(* CoDeSys 2.3.9.48 project: cy-134-wg-002.pro *)
(* Libraries: Standard.lib 8.11.10 12:37:48, SYSLIBCALLBACK.LIB 8.11.10 12:37:48, Ethernet.lib 8.11.10 12:37:48, SysLibEvent.lib 8.11.10 12:37:48, SysLibFile.lib 8.11.10 12:37:48, SysLibPlcCtrl.lib 8.11.10 12:37:48, SysLibRtc.lib 8.11.10 12:37:48, SysLibSockets.lib 5.5.11 09:22:24, Util.lib 26.9.14 11:12:46, Visual.lib 8.11.10 12:37:48, WagoLibIdent.lib 25.2.13 13:49:34, WagoLibMBX_01.lib 20.3.12 16:32:38, WagoLibModbus_IP_01.lib 26.5.15 11:20:08, WagoLibStatus.lib 8.11.10 12:37:48 *)

(* PLC configuration (modules and I/O channels)
VPN_ST AT %IX0.0 [BOOLOnX_I] I 1: Digital Input
LAMP_AL AT %QX0.0 [BOOLOnX_Q] I 2: Digital Input
KEY_QE_ST AT %IX0.1 [BOOLOnX_I] I 3: Digital Input
AT %QX0.1 [BOOLOnX_Q] I 4: Digital Input
AT %IX0.2 [BOOLOnX_I] I 5: Digital Input
AT %QX0.2 [BOOLOnX_Q] I 6: Digital Input
AT %IX0.3 [BOOLOnX_I] I 7: Digital Input
AT %QX0.3 [BOOLOnX_Q] I 8: Digital Input
AT %IX0.4 [BOOLOnX_I] O 1: Digital Output
AT %QX0.4 [BOOLOnX_Q] O 2: Digital Output
AT %IX0.5 [BOOLOnX_I] O 3: Digital Output
AT %QX0.5 [BOOLOnX_Q] O 4: Digital Output
AT %IX0.6 [BOOLOnX_I] O 5: Digital Output
AT %QX0.6 [BOOLOnX_Q] O 6: Digital Output
AT %IX0.7 [BOOLOnX_I] O 7: Digital Output
AT %QX0.7 [BOOLOnX_Q] O 8: Digital Output
Fieldbus variables [FB_VARS] node 1, in %IB0 out %QB0
*)

(* Task configuration *)
TASK PLC_PRG (PRIORITY := 1); (* freewheeling *)
	PLC_PRG();
END_TASK
TASK BACnet (PRIORITY := 2, INTERVAL := T#3000ms);
	PLC_BAC();
END_TASK

(* Global variable list: Global_Constants *)
VAR_GLOBAL CONSTANT

	Plant_NAME			: STRING :='cySN:134 cyVER: Lettura sistema Desigo Ospedale Gavezzeni ';
	Plant_SN			: DWORD  :=134;	(* S/N Impianto di telecontrollo *)
	Plant_SW_VER		: WORD   :=1;		(* Versione SW installata *)


	(* Colour defines *)
	COLOR_RED			: DWORD	:= 16#2020F0;
	COLOR_YELLOW		: DWORD	:= 16#20F0F0;
	COLOR_GREEN			: DWORD	:= 16#20F020;
	COLOR_LIGHT_GREEN	: DWORD := 16#006000;

	(* Parameters *)
(*	Plant_DefaultTAmb	: INT	:=100;		(* [.1°C] Temperatura ambiente di default in caso di rottura sonda *)
	Plant_MaxRunTAmb	: INT   :=210; 		(* [.1°C] Temperatura ambiente massima funzionamento impianto *)
	Plant_AntiFreezeTAmb: INT   :=-40;		(* [.1°C] Antifreeze temperature, start circulators *)
	Plant_VRD_TAlarm	: INT   :=850; 		(* [.1°C] Temperatura di allarme VRD, blocco *)
	Plant_VRD_TMax		: INT   :=800; 		(* [.1°C] Setpoint massimo per uscita VRD *)
	Plant_VRD_TDefault	: INT	:=300;		(* [.1°C] Temperatura di default in caso di errore climatica *)
	Plant_CirOffDelay	: TIME	:=T#30m;	(* (Def.T#15m) Ritardo spegnimento pompe per ricircolo caldaia *)
	Plant_CirOnDelay	: TIME	:=T#15m;
	Plant_MaxWaterLoss	: WORD  :=2;		(* [lt/h] Massima perdita del circuito *) *)

	(* Filesystem *)
	FilesPath  			: STRING :='S:\';

	(* TCP Logger *)
	Logger_SERVER		: STRING:='';
	Logger_IP			: STRING:='10.36.201.146'; (* '192.168.100.3';*)
	Logger_PORT			: WORD  :=80;
	Logger_GETSTART		: STRING:='GET /cygmsrv/hsgm.ashx?';
	Logger_GETEND		: STRING:='$R$N$R$N';
	Logger_CHECK		: STRING:='True';
	Logger_CRLF			: STRING:='$R$N';
	Logger_DataFile		: STRING:='S:\LOG.DAT';
	Logger_DataFileOld	: STRING:='S:\LOG.BCK';
	Logger_IndexFile	: STRING:='S:\LOG.IDX';
	Logger_ConnRetries	: BYTE:=5;
	Logger_RecoverMsgs	: BYTE:=25;

	(* TCP Remote *)
	Remote_PORT			: WORD  :=10;
	Remote_WELCOME		: STRING:='Connected$R$N';
	Remote_OK			: STRING:='OK$R$N';
	Remote_ERROR		: STRING:='ERROR$R$N';

	(* TCP Sockets *)
	MAX_SEND_TCP_SERVER					 : DWORD:=30000;(*60000*)
	MAX_RECEIVE_TCP_SERVER				 : DWORD:=3000;
	MAX_RECEIVE_TCP_SERVER_SOCKET	 	 : DWORD:=1500;
	MAX_SEND_TCP_CLIENT					 : DWORD:=30000;(*15000*)
	MAX_RECEIVE_TCP_CLIENT				 : DWORD:=1500;
	MAX_RECEIVE_TCP_CLIENT_SOCKET		 : DWORD:=1500;
	MAX_RECEIVE_UDP_SERVER				 : INT  :=1472;
	MAX_RECEIVE_UDP_CLIENT				 : INT  :=1472;
	CONNECT_WATCHDOG_TIME				 : TIME :=t#10s;

END_VAR

(* Global variable list: Global_Variables *)
VAR_GLOBAL

	SYS    : typ_SYS;
	Logger : typ_Logger;


	Lamp	:	LAMP_AL_GENERALE;

	(* Analizzatori presenti  *)
	ANZ01  : obj_ANZ_Recupero_01	:= ( ID:=1 , ContabilizerMode:=0);     	(* Generale  QE1  -  Sottorete OP11 - BsB_Mulcab4_Cab4QE1 *)
	ANZ02  : obj_ANZ_Recupero_01	:= ( ID:=2 , ContabilizerMode:=0);		(* Generale  QE2 Continità - Sottorete OP11  - BsB_MulCab4_Cab4QE2C *)
	ANZ03  : obj_ANZ_Recupero_01	:= ( ID:=3 , ContabilizerMode:=0);		(* Generale  QE2  - Sottorete OP11  - BsB_MulCab4_Cab4QE2P *)
	ANZ04  : obj_ANZ_Recupero_01	:= ( ID:=4 , ContabilizerMode:=0);		(* Gruppo  Frigorifero CHW01  - Sottorete OP22  - Mult_MulC_QEGF01 *)
	ANZ05  : obj_ANZ_Recupero_01	:= ( ID:=5 , ContabilizerMode:=0);		(* Gruppo Frigorifero CHW-02 - Sottorette OP22 - Mult_MulC_QGGF02 *)
	ANZ06  : obj_ANZ_Recupero_01	:= ( ID:=6 , ContabilizerMode:=0);		(* Generale da trafo TR1 - Sottorette OP22 - Mult_QGBT02 *)
	ANZ07  : obj_ANZ_Recupero_01	:= ( ID:=7 , ContabilizerMode:=0);		(* Alimentazione Piastra 1 da QGBT - OP22 - Mult_QGBT03 *)
	ANZ08  : obj_ANZ_Recupero_01	:= ( ID:=8 , ContabilizerMode:=0);		(* Generale da trafo TR3 - OP22 - Mult_QGBT04 *)
	ANZ09  : obj_ANZ_Recupero_01	:= ( ID:=9 , ContabilizerMode:=0);		(* Gruppo frigo GF01 - OP22 - Mult_QGBT07 *)
	ANZ10  : obj_ANZ_Recupero_01	:= ( ID:=10 , ContabilizerMode:=0);	(* Riserva futuro frigorifero - OP22 - Mult_QGBT08 *)
	ANZ11  : obj_ANZ_Recupero_01	:= ( ID:=11 , ContabilizerMode:=0);	(* Riserva - OP22 - Mult_QGBT09 *)
	ANZ12  : obj_ANZ_Recupero_01	:= ( ID:=12 , ContabilizerMode:=0);	(* Riserva - OP22 - Mult_QGBT10 *)
	ANZ13  : obj_ANZ_Recupero_01	:= ( ID:=13 , ContabilizerMode:=0);	(* Impianto Water Mist - OP22 - Mult_QGBT11 *)
	ANZ14  : obj_ANZ_Recupero_01	:= ( ID:=14 , ContabilizerMode:=0);	(* QP3 Piano terzo D - OP22 - Mult_QGBT12 *)
	ANZ15  : obj_ANZ_Recupero_01	:= ( ID:=15 , ContabilizerMode:=0);	(* QP2 Piano secondo D - OP22 - Mult_QGBT13 *)
	ANZ16  : obj_ANZ_Recupero_01	:= ( ID:=16 , ContabilizerMode:=0);	(* QP1 Piano primo D - OP22 - Mult_QGBT14 *)
	ANZ17  : obj_ANZ_Recupero_01	:= ( ID:=17 , ContabilizerMode:=0);	(* QPT Piano terra D - OP22 - Mult_QGBT15 *)
	ANZ18  : obj_ANZ_Recupero_01	:= ( ID:=18 , ContabilizerMode:=0);	(* QPI Piano interrato D - OP22 - Mult_QGBT16 *)
	ANZ19  : obj_ANZ_Recupero_01	:= ( ID:=19 , ContabilizerMode:=0);	(* Alimentazione cabina ricevimento L1 - OP22 - Mult_QGBT17 *)
	ANZ20  : obj_ANZ_Recupero_01	:= ( ID:=20 , ContabilizerMode:=0);	(* Alimentazione cabina ricevimento L2 - OP22 - Mult_QGBT18 *)
	ANZ21  : obj_ANZ_Recupero_01	:= ( ID:=21 , ContabilizerMode:=0);	(*  Sezione generale da UPS1 - OP22 - Mult_QUPS01 *)
	ANZ22  : obj_ANZ_Recupero_01	:= ( ID:=22 , ContabilizerMode:=0);	(*  Sezione generale - OP22 - Mult_QUPS02 *)
	ANZ23  : obj_ANZ_Recupero_01	:= ( ID:=23 , ContabilizerMode:=0);	(*  Sezione generale da UPS2 - OP22 - Mult_QUPS03 *)
	ANZ24  : obj_ANZ_Recupero_01	:= ( ID:=24 , ContabilizerMode:=0);	(*  QP3 sezione dialisi - OP22 - Mult_QUPS04 *)
	ANZ25  : obj_ANZ_Recupero_01	:= ( ID:=25 , ContabilizerMode:=0);
	ANZ26  : obj_ANZ_Recupero_01	:= ( ID:=26 , ContabilizerMode:=0);	(* Generale Villa Elios- OP23 - Mult1'QEPC_QUPS0 *)
	ANZ27  : obj_ANZ_Recupero_01	:= ( ID:=27 , ContabilizerMode:=0);	(*Generale sez. preferenziale - OP23 - Mult1_ QGBT05*)
	ANZ28  : obj_ANZ_Recupero_01	:= ( ID:=28 , ContabilizerMode:=0);	(* generale G.E. - OP23 - Mult1'QGBT06 *)
	ANZ29  : obj_ANZ_Recupero_01	:= ( ID:=29 , ContabilizerMode:=0);	(* Gruppo frigo polivalente GP01 - OP23 - Mult1_QGBT19 *)
	ANZ30  : obj_ANZ_Recupero_01	:= ( ID:=30 , ContabilizerMode:=0);	(*QP2 quadro piano 2 - OP23 - Mul1_QGBT20*)
	ANZ31  : obj_ANZ_Recupero_01	:= ( ID:=31 , ContabilizerMode:=0);	(*QP1 quadro piano 1 - OP23 - Mult1_QGBT21*)
	ANZ32  : obj_ANZ_Recupero_01	:= ( ID:=32 , ContabilizerMode:=0);	(*QPT quadro piano terra - OP23 - Mult1_QGBT22*)
	ANZ33  : obj_ANZ_Recupero_01	:= ( ID:=33 , ContabilizerMode:=0);	(*QPI quadro piano interrato - OP23 - Mult1_QGBT23*)
	ANZ34  : obj_ANZ_Recupero_01	:= ( ID:=34 , ContabilizerMode:=0);	(*QP3 quadro piano terzo - OP23 - Mult1_QGBT24*)
	ANZ35  : obj_ANZ_Recupero_01	:= ( ID:=35 , ContabilizerMode:=0);	(*Quadro centrale UTA copertura - OP23 - Mult1_QGBT25*)
	ANZ36  : obj_ANZ_Recupero_01	:= ( ID:=36 , ContabilizerMode:=0);	(*Quadro centrale UTA esterno PT - OP23 - Mult1_QGBT26*)
	ANZ37  : obj_ANZ_Recupero_01	:= ( ID:=37 , ContabilizerMode:=0);	(*Quadro centrale idrica interrato - OP23 - Mult1_QGBT27*)
	ANZ38  : obj_ANZ_Recupero_01	:= ( ID:=38 , ContabilizerMode:=0);	(*Riserva - OP23 - Mult1_QGBT28*)
	ANZ39  : obj_ANZ_Recupero_01	:= ( ID:=39 , ContabilizerMode:=0);	(*Nuova TAC - OP23 - Mult1_QGBT29*)
	ANZ40  : obj_ANZ_Recupero_01	:= ( ID:=40 , ContabilizerMode:=0);	(*UPS1 - OP23 - Mult1_QGBT30*)
	ANZ41  : obj_ANZ_Recupero_01	:= ( ID:=41 , ContabilizerMode:=0);	(*UPS2 - OP23 - Mult1_QGBT31*)
	ANZ42  : obj_ANZ_Recupero_01	:= ( ID:=42 , ContabilizerMode:=0);	(*by-pass UPS1 - OP23 - Mult1_QGBT32*)
	ANZ43  : obj_ANZ_Recupero_01	:= ( ID:=43 , ContabilizerMode:=0);	(*by-pass UPS2 - OP23 - Mult1_QGBT33*)
	ANZ44  : obj_ANZ_Recupero_01	:= ( ID:=44 , ContabilizerMode:=0);	(*by-pass di sistema - OP23 - Mult1_QGBT34*)
	ANZ45  : obj_ANZ_Recupero_01	:= ( ID:=45 , ContabilizerMode:=0);	(*Quadro centrale termofrigorifera- OP23 - Mult1_QGBT35*)
	ANZ46  : obj_ANZ_Recupero_01	:= ( ID:=46 , ContabilizerMode:=0);			(* Gruppo Frigorifero CHW-03 - Sottorette OP22 - Mult_MulC_QGGF03 *)
	ANZ47  : obj_ANZ_Recupero_01	:= ( ID:=47 , ContabilizerMode:=0);			(* Alimentazione Piastra 1 da trafo TR1 - Sottorette OP22 - Mult_QGBT01 *)









END_VAR


VAR_GLOBAL CONSTANT


	MAX_Weekly_Schedule							: BYTE:=7;		(*Parameter for BACNET_SCHEDULE Object*)
	MAX_Exception_Schedule						: BYTE:=7;		(*Parameter for BACNET_SCHEDULE Object*)
	MAX_List_Of_Object_Property_References		: BYTE:=7;		(*Parameter for BACNET_SCHEDULE Object*)


	MAX_DateList								: BYTE:=14;	(*Parameter for BACNET_CALENDAR Object*)
	MAX_DeviceAddressBinding					: BYTE:=7;		(*Parameter for BACNET_DEVICE Object*)
	MAX_Configuration_Files						: BYTE:=4;		(*Parameter for BACNET_DEVICE Object*)
	MAX_Active_COV_Subscriptions				: BYTE:=7;		(*Parameter for BACNET_DEVICE Object*)
	MAX_List_Of_Group_Members					: BYTE:=7;		(*Parameter for BACNET_GROUP Object*)
	MAX_Accepted_Modes							: BYTE := 15;	(*Parameter for BACNET_LIFE_SAFETY_POINT / ZONE Object*)
	MAX_Life_Safety_Alarm_Values				: BYTE := 24;	(*Parameter for BACNET_LIFE_SAFETY_POINT / ZONE Object*)
	MAX_Alarm_Values							: BYTE := 24;	(*Parameter for BACNET_LIFE_SAFETY_POINT / ZONE Object*)
	MAX_Fault_Values							: BYTE := 24;	(*Parameter for BACNET_LIFE_SAFETY_POINT / ZONE Object*)
	MAX_Member_Of								: BYTE := 3;	(*Parameter for BACNET_LIFE_SAFETY_POINT / ZONE Object*)
	MAX_Zone_Members							: BYTE := 3;	(*Parameter for BACNET_LIFE_SAFETY_ ZONE Object*)
	MAX_State_Text								: BYTE:=24;	(*Parameter for BACNET_MULTISTATE_VALUE Object*)
	MAX_Alarm_Values_1							: BYTE:=24;	(*Parameter for BACNET_MULTISTATE_VALUE Object*)
	MAX_Fault_Values_1							: BYTE := 24;	(*Parameter for BACNET_MULTISTATE_VALUE Object*)
	MAX_Recipient_List							: BYTE:=8;		(*Parameter for BACNET_NOTIFICATION_CLASS Object*)
	MAX_Log_Buffer								: BYTE:=24;	(*Parameter for BACNET_TREND_LOG Object*)
	MAX_listOfPropertyReferences				: BYTE:=7;		(*Parameter for ReadAccessSpecification data type*)
END_VAR

(* Data type in Enumerationen *)
TYPE AccumulatorStatus :(
	normal_1	:=0,
	starting	:=1,
	recovered	:=2,
	abnormal	:=3,
	failed		:=4);
END_TYPE

(* Data type in Objects *)
TYPE BACNET_ACCUMULATOR :
STRUCT
	Object_Identifier			:BACnetObjectIdentifier;
	Object_Name				:STRING(48);
	Object_Type				:BACnetObjectType;
	Present_Value			:WORD;
	Description				:STRING(48);
	Device_Type				:STRING(48);
	Status_Flags				:BACnetStatusFlags;
	Event_State				:BACnetEventState;
	Reliability					:BACnetReliability;
	Out_Of_Service			:BOOL;
	Scale						:BACnetScale;
	Units						:BACnetEngineeringUnits;
	Prescale					:BACnetPrescale;
	Max_Pres_Value			:WORD;
	Value_Change_Time		:BACnetDateTime;
	Value_Before_Change	:WORD;
	Value_Set					:WORD;
	Pulse_Rate				:WORD;
	High_Limit				:WORD;
	Low_Limit					:WORD;
	Limit_Monitoring_Interval	:WORD;
	Notification_Class		:WORD;
	Time_Delay				:WORD;
	Limit_Enable				:BACnetLimitEnable;
	Event_Enable				:BACnetEventTransitionBits;
	Acked_Transitions		:BACnetEventTransitionBits;
	Notify_Type				:BACnetNotifyType;
	Event_Time_Stamps		:ARRAY [1..3] OF BACnetTimeStamp;
END_STRUCT
END_TYPE

(* Data type in Objects *)
TYPE BACNET_ANALOG_INPUT :
STRUCT
 	Object_Identifier			:BACnetObjectIdentifier;
	Object_Name				:STRING(48);
	Object_Type				:BACnetObjectType;
	Present_Value			:REAL;
	Description				:STRING(48);
	Device_Type				:STRING(48);
	Status_Flags				:BACnetStatusFlags;
	Event_State				:BACnetEventState;
	Reliability					:BACnetReliability;
	Out_of_Service			:BOOL;
	Update_Interval			:WORD;
	Units						:BACnetEngineeringUnits;
	COV_Increment			:REAL;
	Time_Delay				:WORD;
	Notification_Class		:WORD;
	High_Limit				:REAL;
	Low_Limit					:REAL;
	Deadband					:REAL;
	Limit_Enable				:BACnetLimitEnable;
	Event_Enable				:BACnetEventTransitionBits;
	Acked_Transitions		:BACnetEventTransitionBits;
	Notify_Type				:BACnetNotifyType;
	Event_Time_Stamps		:ARRAY [1..3] OF BACnetTimeStamp;
END_STRUCT
END_TYPE

(* Data type in Objects *)
TYPE BACNET_ANALOG_OUTPUT :
STRUCT
	Object_Identifier		:BACnetObjectIdentifier;
	Object_Name			:STRING(48);
	Object_Type			:BACnetObjectType;
	Present_Value		:REAL;
	Description			:STRING(48);
	Device_Type			:STRING(48);
	Status_Flags			:BACnetStatusFlags;
	Event_State			:BACnetEventState;
	Reliability				:BACnetReliability;
	Out_Of_Service		:BOOL;
	Units					:BACnetEngineeringUnits;
	Priority_Array			:BACnetPriorityArray;
	Relinquish_Default	:REAL;
	COV_Increment		:REAL;
	Time_Delay			:WORD;
	Notification_Class	:WORD;
	High_Limit			:REAL;
	Low_Limit				:REAL;
	Deadband				:REAL;
	Limit_Enable			:BACnetLimitEnable;
	Event_Enable			:BACnetEventTransitionBits;
	Acked_Transitions	:BACnetEventTransitionBits;
	Notify_Type			:BACnetNotifyType;
	Event_Time_Stamps	:ARRAY [1..3] OF BACnetTimeStamp;
END_STRUCT
END_TYPE

(* Data type in Objects *)
TYPE BACNET_ANALOG_VALUE :
STRUCT
	Object_Identifier		:BACnetObjectIdentifier;
	Object_Name			:STRING(48);
	Object_Type			:BACnetObjectType;
	Present_Value		:REAL;
	Description			:STRING(48);
	Status_Flags			:BACnetStatusFlags;
	Event_State			:BACnetEventState;
	Reliability				:BACnetReliability;
	Out_Of_Service		:BOOL;
	Units					:BACnetEngineeringUnits;
	Priority_Array			:ARRAY [1..16] OF REAL;
	Relinquish_Default	:REAL;
	COV_Increment		:REAL;
	Time_Delay			:WORD;
	Notification_Class	:WORD;
	High_Limit			:REAL;
	Low_Limit				:REAL;
	Deadband				:REAL;
	Limit_Enable			:BACnetLimitEnable;
	Event_Enable			:BACnetEventTransitionBits;
	Acked_Transitions	:BACnetEventTransitionBits;
	Notify_Type			:BACnetNotifyType;
	Event_Time_Stamps	:ARRAY [1..3] OF BACnetTimeStamp;
END_STRUCT
END_TYPE

(* Data type in Objects *)
TYPE BACNET_AVERAGING :
STRUCT
 	Object_Identifier				:BACnetObjectIdentifier;
	Object_Name					:STRING(48);
	Object_Type					:BACnetObjectType;
	Minimum_Value				:REAL;
	Minimum_Value_Timestamp:BACnetDateTime;
	Average_Value				:REAL;
	Variance_Value				:REAL;
	Maximum_Value				:REAL;
	Maximum_Value_Timestamp:BACnetDateTime;
	Description					:STRING(48);
	Attempted_Samples			:WORD;
	Valid_Samples				:WORD;
	Object_Property_Reference	:BACnetDeviceObjectPropertyReference;
	Window_Interval				:WORD;
	Window_Samples			:WORD;
END_STRUCT
END_TYPE

(* Data type in Objects *)
TYPE BACNET_BINARY_INPUT :
STRUCT
	Object_Identifier				:BACnetObjectIdentifier;
	Object_Name					:STRING(48);
	Object_Type					:BACnetObjectType;
	Present_Value				:BACnetBinaryPV;
	Description					:STRING(48);
	Device_Type					:STRING(48);
	Status_Flags					:BACnetStatusFlags;
	Event_State					:BACnetEventState;
	Reliability						:BACnetReliability;
	Out_Of_Service				:BOOL;
	Polarity						:BACnetPolarity;
	Inactive_Text					:STRING(48);
	Active_Text					:STRING(48);
	Change_Of_State_Time		:BACnetDateTime;
	Change_Of_State_Count		:WORD;
	Time_Of_State_Count_Reset:BACnetDateTime;
	Elapsed_Active_Time			:DWORD;
	Time_Of_Active_Time_Reset:BACnetDateTime;
	Time_Delay					:WORD;
	Notification_Class			:WORD;
	Alarm_Value					:BACnetBinaryPV;
	Event_Enable					:BACnetEventTransitionBits;
	Acked_Transitions			:BACnetEventTransitionBits;
	Notify_Type					:BACnetNotifyType;
	Event_Time_Stamps			:ARRAY [1..3] OF BACnetTimeStamp;
END_STRUCT
END_TYPE

(* Data type in Objects *)
TYPE BACNET_BINARY_OUTPUT :
STRUCT
 Object_Identifier					:BACnetObjectIdentifier;
 Object_Name						:STRING(48);
 Object_Type						:BACnetObjectType;
 Present_Value					:BACnetBinaryPV;
 Description						:STRING(48);
 Device_Type						:STRING(48);
 Status_Flags						:BACnetStatusFlags;
 Event_State						:BACnetEventState;
 Reliability							:BACnetReliability;
 Out_Of_Service					:BOOL;
 Polarity							:BACnetPolarity;
 Inactive_Text						:STRING(48);
 Active_Text						:STRING(48);
 Change_Of_State_Time			:BACnetDateTime;
 Change_Of_State_Count		:WORD;
 Time_Of_State_Count_Reset	:BACnetDateTime;
 Elapsed_Active_Time			:DWORD;
 Time_Of_Active_Time_Reset	:BACnetDateTime;
 Minimum_Off_Time				:DWORD;
 Minimum_On_Time				:DWORD;
 Priority_Array						:BACnetPriorityArray;
 Relinquish_Default				:BACnetBinaryPV;
 Time_Delay						:WORD;
 Notification_Class				:WORD;
 Feedback_Value					:BACnetBinaryPV;
 Event_Enable						:BACnetEventTransitionBits;
 Acked_Transitions				:BACnetEventTransitionBits;
 Notify_Type						:BACnetNotifyType;
 Event_Time_Stamps				:ARRAY [1..3] OF BACnetTimeStamp;
END_STRUCT
END_TYPE

(* Data type in Objects *)
TYPE BACNET_BINARY_VALUE :
STRUCT
	Object_Identifier					:BACnetObjectIdentifier;
	Object_Name						:STRING(48);
	Object_Type						:BACnetObjectType;
	Present_Value					:BACnetBinaryPV;
	Description						:STRING(48);
	Status_Flags						:BACnetStatusFlags;
	Event_State						:BACnetEventState;
	Reliability							:BACnetReliability;
	Out_Of_Service					:BOOL;
	Inactive_Text						:STRING(48);
	Active_Text						:STRING(48);
	Change_Of_State_Time			:BACnetDateTime;
	Change_Of_State_Count			:DWORD;
	Time_Of_State_Count_Reset	:BACnetDateTime;
	Elapsed_Active_Time				:DWORD;
	Time_Of_Active_Time_Reset	:BACnetDateTime;
	Minimum_Off_Time				:DWORD;
	Minimum_On_Time				:DWORD;
	Priority_Array						:ARRAY [1..16] OF BACnetBinaryPV;
	Relinquish_Default				:BACnetBinaryPV;
	Time_Delay						:WORD;
	Notification_Class				:WORD;
	Alarm_Value						:BACnetBinaryPV;
	Event_Enable						:BACnetEventTransitionBits;
	Acked_Transitions				:BACnetEventTransitionBits;
	Notify_Type						:BACnetNotifyType;
	Event_Time_Stamps				:ARRAY [1..3] OF BACnetTimeStamp;
END_STRUCT
END_TYPE

(* Data type in Objects *)
TYPE BACNET_CALENDAR :
STRUCT
	Object_Identifier		:BACnetObjectIdentifier;
	Object_Name			:STRING(48);
	Object_Type			:BACnetObjectType;
	Description			:STRING(48);
	Present_Value		:BOOL;
	Date_List				:ARRAY[0..MAX_DateList] OF BACnetCalendarEntry;
END_STRUCT
END_TYPE

(* Data type in Objects *)
TYPE BACNET_COMMAND :
STRUCT
	Object_Identifier			:BACnetObjectIdentifier;
	Object_Name				:STRING(48);
	Object_Type				:BACnetObjectType;
	Description				:STRING(48);
	Present_Value			:WORD;
	In_Process				:BOOL;
	All_Writes_Successful	:BOOL;
	Action_					:ARRAY [1..3] OF BACnetActionList;
	Action_Text				:ARRAY [1..3] OF STRING(48);
END_STRUCT
END_TYPE

(* Data type in Objects *)
TYPE BACNET_DEVICE :
STRUCT
	Object_Identifier						:BACnetObjectIdentifier;
	Object_Name							:STRING(48);
	Object_Type							:BACnetObjectType;
	System_Status						:BACnetDeviceStatus;
	Vendor_Name						:STRING(48);
	Vendor_Identifier						:WORD;
	Model_Name							:STRING(48);
	Firmware_Revision					:STRING(48);
	Application_Software_Version		:STRING(48);
	Location								:STRING(48);
	Description							:STRING(48);
	Protocol_Version						:WORD;
	Protocol_Revision					:WORD;
	Protocol_Services_Supported		:BACnetServicesSupported;
	Protocol_Object_Types_Supported	:BACnetObjectTypesSupported;
	Object_List							:ARRAY [1..3] OF BACnetObjectIdentifier;
	Max_APDU_Length_Accepted		:WORD;
	Segmentation_Supported			:BACnetSegmentation;
	Max_Segments_Accepted			:WORD;
	Local_Time							:TIME;
	Local_Date							:DATE;
	UTC_Offset							:INT;
	Daylight_Savings_Status				:BOOL;
	APDU_Segment_Timeout			:WORD;
	APDU_Timeout						:WORD;
	Number_Of_APDU_Retries			:WORD;
	Device_Address_Binding				:ARRAY [0..MAX_DeviceAddressBinding] OF BACnetAddressBinding;
	Database_Revision					:WORD;
	Configuration_Files					:ARRAY [1..MAX_Configuration_Files] OF BACnetObjectIdentifier;
	Last_Restore_Time					:BACnetTimeStamp;
	Backup_Failure_Timeout				:WORD;
	Active_COV_Subscriptions			:ARRAY [0..MAX_Active_COV_Subscriptions] OF BACnetCOVSubscription;
END_STRUCT
END_TYPE

(* Data type in Objects *)
TYPE BACNET_EVENT_ENROLLMENT :
STRUCT
	Object_Identifier				:BACnetObjectIdentifier;
	Object_Name					:STRING(48);
	Object_Type					:BACnetObjectType;
	Description					:STRING(48);
	Event_Type					:BACnetEventType;
	Notify_Type					:BACnetNotifyType;
	Event_Parameters			:BACnetEventParameter;
	Object_Property_Reference	:BACnetDeviceObjectPropertyReference;
	Event_State					:BACnetEventState;
	Event_Enable					:BACnetEventTransitionBits;
	Acked_Transitions			:BACnetEventTransitionBits;
	Notification_Class			:WORD;
	Event_Time_Stamps			:ARRAY [1..3] OF BACnetTimeStamp;
END_STRUCT
END_TYPE

(* Data type in Objects *)
TYPE BACNET_FILE :
STRUCT
	Object_Identifier		:BACnetObjectIdentifier;
	Object_Name			:STRING(48);
	Object_Type			:BACnetObjectType;
	Description			:STRING(48);
	File_Type				:STRING(48);
	File_Size				:WORD;
	Modification_Date		:BACnetDateTime;
	Archive					:BOOL;
	Read_Only_			:BOOL;
	File_Access_Method	:BACnetFileAccessMethod;
END_STRUCT
END_TYPE

(* Data type in Objects *)
TYPE BACNET_GROUP :
STRUCT
	Object_Identifier			:BACnetObjectIdentifier;
	Object_Name				:STRING(48);
	Object_Type				:BACnetObjectType;
	Description				:STRING(48);
	List_Of_Group_Members	:ARRAY [0..MAX_List_Of_Group_Members] OF ReadAccessSpecification;
	Present_Value			:ARRAY [0..MAX_List_Of_Group_Members] OF ReadAccessResult;
END_STRUCT
END_TYPE

(* Data type in Objects *)
TYPE BACNET_LIFE_SAFETY_POINT :
STRUCT
	Object_Identifier				:BACnetObjectIdentifier;
	Object_Name					:STRING(48);
	Object_Type					:BACnetObjectType;
	Present_Value				:BACnetLifeSafetyState;
	Tracking_Value				:BACnetLifeSafetyState;
	Description					:STRING(48);
	Device_Type					:STRING(48);
	Status_Flags					:BACnetStatusFlags;
	Event_State					:BACnetEventState;
	Reliability						:BACnetReliability;
	Out_Of_Service				:BOOL;
	Mode							:BACnetLifeSafetyMode;
	Accepted_Modes				:ARRAY [0..MAX_Accepted_Modes] OF BACnetLifeSafetyMode;
	Time_Delay					:WORD;
	Notification_Class			:WORD;
	Life_Safety_Alarm_Values	:ARRAY  [0..MAX_Life_Safety_Alarm_Values]  OF BACnetLifeSafetyState;
	Alarm_Values					:ARRAY  [0..MAX_Alarm_Values]  OF BACnetLifeSafetyState;
	Fault_Values					:ARRAY  [0..MAX_Fault_Values]  OF BACnetLifeSafetyState;
	Event_Enable					:BACnetEventTransitionBits;
	Acked_Transitions			:BACnetEventTransitionBits;
	Notify_Type					:BACnetNotifyType;
	Event_Time_Stamps			:ARRAY [1..3] OF BACnetTimeStamp;
	Silenced						:BACnetSilencedState;
	Operation_Expected			:BACnetLifeSafetyOperation;
	Maintenance_Required		:BACnetMaintenance;
	Setting							:BYTE;
	Direct_Reading				:REAL;
	Units							:BACnetEngineeringUnits;
	Member_Of					:ARRAY [1..MAX_Member_Of]  OF BACnetDeviceObjectReference;
END_STRUCT
END_TYPE

(* Data type in Objects *)
TYPE BACNET_LIFE_SAFETY_ZONE :
STRUCT
	Object_Identifier				:BACnetObjectIdentifier;
	Object_Name					:STRING(48);
	Object_Type					:BACnetObjectType;
	Present_Value				:BACnetLifeSafetyState;
	Tracking_Value				:BACnetLifeSafetyState;
	Description					:STRING(48);
	Device_Type					:STRING(48);
	Status_Flags					:BACnetStatusFlags;
	Event_State					:BACnetEventState;
	Reliability						:BACnetReliability;
	Out_Of_Service				:BOOL;
	Mode							:BACnetLifeSafetyMode;
	Accepted_Modes				:ARRAY  [0..MAX_Accepted_Modes] OF BACnetLifeSafetyMode;
	Time_Delay					:WORD;
	Notification_Class			:WORD;
	Life_Safety_Alarm_Values	:ARRAY [0..MAX_Life_Safety_Alarm_Values] OF BACnetLifeSafetyState;
	Alarm_Values					:ARRAY [0..MAX_Alarm_Values] OF BACnetLifeSafetyState;
	Fault_Values					:ARRAY [0..MAX_Fault_Values] OF BACnetLifeSafetyState;
	Event_Enable					:BACnetEventTransitionBits;
	Acked_Transitions			:BACnetEventTransitionBits;
	Notify_Type					:BACnetNotifyType;
	Event_Time_Stamps			:ARRAY [1..3] OF BACnetTimeStamp;
	Silenced						:BACnetSilencedState;
	Operation_Expected			:BACnetLifeSafetyOperation;
	Maintenance_Required		:BOOL;
	Zone_Members				:ARRAY [1..MAX_Zone_Members] OF BACnetDeviceObjectReference;
	Member_Of					:ARRAY [1..MAX_Member_Of] OF BACnetDeviceObjectReference;
END_STRUCT
END_TYPE

(* Data type in Objects *)
TYPE BACNET_LOOP :
STRUCT
	Object_Identifier						:BACnetObjectIdentifier;
	Object_Name							:STRING(48);
	Object_Type							:BACnetObjectType;
	Present_Value						:REAL;
	Description							:STRING(48);
	Status_Flags							:BACnetStatusFlags;
	Event_State							:BACnetEventState;
	Reliability								:BACnetReliability;
	Out_Of_Service						:BOOL;
	Update_Interval						:WORD;
	Output_Units							:BACnetEngineeringUnits;
	Manipulated_Variable_Reference	:BACnetObjectPropertyReference;
	Controlled_Variable_Reference		:BACnetObjectPropertyReference;
	Controlled_Variable_Value			:REAL;
	Controlled_Variable_Units			:BACnetEngineeringUnits;
	Setpoint_Reference					:BACnetSetpointReference;
	Setpoint								:REAL;
	ACTION_								:BACnetAction;
	Proportional_Constant				:REAL;
	Proportional_Constant_Units		:BACnetEngineeringUnits;
	Integral_Constant						:REAL;
	Integral_Constant_Units				:BACnetEngineeringUnits;
	Derivative_Constant					:REAL;
	Derivative_Constant_Units			:BACnetEngineeringUnits;
	Bias									:REAL;
	Maximum_Output						:REAL;
	Minimum_Output						:REAL;
	Priority_For_Writing					:WORD;
	COV_Increment						:REAL;
	Time_Delay							:WORD;
	Notification_Class					:WORD;
	Error_Limit							:REAL;
	Event_Enable							:BACnetEventTransitionBits;
	Acked_Transitions					:BACnetEventTransitionBits;
	Notify_Type							:BACnetNotifyType;
	Event_Time_Stamps					:ARRAY [1..3] OF BACnetTimeStamp;
END_STRUCT
END_TYPE

(* Data type in Objects *)
TYPE BACNET_MULTISTATE_VALUE :
STRUCT
	Object_Identifier		:BACnetObjectIdentifier;
	Object_Name			:STRING(48);
	Object_Type			:BACnetObjectType;
	Present_Value		:WORD;
	Description			:STRING(48);
	Status_Flags			:BACnetStatusFlags;
	Event_State			:BACnetEventState;
	Reliability				:BACnetReliability;
	Out_Of_Service		:BOOL;
	Number_Of_States	:WORD;
	State_Text				:ARRAY [1..MAX_State_Text] OF STRING(48);
	Priority_Array			:BACnetPriorityArray;
	Relinquish_Default	:WORD;
	Time_Delay			:WORD;
	Notification_Class	:WORD;
	Alarm_Values			:ARRAY [1..MAX_Alarm_Values_1] OF WORD;
	Fault_Values			:ARRAY [1..MAX_Fault_Values_1] OF WORD;
	Event_Enable			:BACnetEventTransitionBits;
	Acked_Transitions	:BACnetEventTransitionBits;
	Notify_Type			:BACnetNotifyType;
	Event_Time_Stamps	:ARRAY [1..3] OF BACnetTimeStamp;
END_STRUCT
END_TYPE

(* Data type in Objects *)
TYPE BACNET_NOTIFICATION_CLASS :
STRUCT
	Object_Identifier		:BACnetObjectIdentifier;
	Object_Name			:STRING(48);
	Object_Type			:BACnetObjectType;
	Description			:STRING(48);
	Notification_Class	:WORD;
	Priority					:ARRAY [1..3] OF WORD;
	Ack_Required			:BACnetEventTransitionBits;
	Recipient_List			:ARRAY [0..MAX_Recipient_List] OF BACnetDestination;
END_STRUCT
END_TYPE

(* Data type in Objects *)
TYPE BACNET_PROGRAM :
STRUCT
	Object_Identifier			:BACnetObjectIdentifier;
	Object_Name				:STRING(48);
	Object_Type				:BACnetObjectType;
	Program_State			:BACnetProgramState;
	Program_Change			:BACnetProgramRequest;
	Reason_For_Halt			:BACnetProgramError;
	Description_Of_Halt		:STRING(48);
 	Program_Location		:STRING(48);
	Description				:STRING(48);
	Status_Flags				:BACnetStatusFlags;
	Reliability					:BACnetReliability;
	Out_Of_Service			:BOOL;
END_STRUCT
END_TYPE

(* Data type in Objects *)
TYPE BACNET_PULSE_CONVERTER :
STRUCT
	Object_Identifier			:BACnetObjectIdentifier;
	Object_Name				:STRING(48);
	Object_Type				:BACnetObjectType;
	Description				:STRING(48);
	Present_Value			:REAL;
	Input_Reference			:BACnetObjectPropertyReference;
	Status_Flags				:BACnetStatusFlags;
	Event_State				:BACnetEventState;
	Reliability					:BACnetReliability;
	Out_Of_Service			:BOOL;
	Units						:BACnetEngineeringUnits;
	Scale_Factor				:REAL;
	Adjust_Value				:REAL;
	Count						:WORD;
	Update_Time				:BACnetDateTime;
	Count_Change_Time		:BACnetDateTime;
	Count_Before_Change	:WORD;
	COV_Increment			:REAL;
	COV_Period				:WORD;
	Notification_Class		:WORD;
	Time_Delay				:WORD;
	High_Limit				:REAL;
	Low_Limit					:REAL;
	Deadband					:REAL;
	Limit_Enable				:BACnetLimitEnable;
	Event_Enable				:BACnetEventTransitionBits;
	Acked_Transitions		:BACnetEventTransitionBits;
	Notify_Type				:BACnetNotifyType;
	Event_Time_Stamps		:ARRAY [1..3] OF BACnetTimeStamp;
END_STRUCT
END_TYPE

(* Data type in Objects *)
TYPE BACNET_SCHEDULE :
STRUCT
	Object_Identifier							:BACnetObjectIdentifier;
	Object_Name								:STRING(48);
	Object_Type								:BACnetObjectType;
	Present_Value							:BACnetAny;
	Description								:STRING(48);
	Effective_Period							:BACnetDateRange;
	Weekly_Schedule							:ARRAY [0..MAX_Weekly_Schedule] OF BACnetDailySchedule;
	Exception_Schedule						:ARRAY [0..MAX_Exception_Schedule] OF BACnetSpecialEvent;
	Schedule_Default							:BACnetAny;
	List_Of_Object_Property_References	:ARRAY [0..MAX_List_Of_Object_Property_References] OF BACnetDeviceObjectPropertyReference;
	Priority_For_Writing						:BYTE;
	Status_Flags								:BACnetStatusFlags;
	Reliability									:BACnetReliability;
	Out_Of_Service							:BOOL;
END_STRUCT
END_TYPE

(* Data type in Objects *)
TYPE BACNET_TREND_LOG :
STRUCT
	Object_Identifier				:BACnetObjectIdentifier;
	Object_Name					:STRING(48);
	Object_Type					:BACnetObjectType;
	Description					:STRING(48);
	Log_Enable					:BOOL;
	Start_Time					:BACnetDateTime;
	Stop_Time					:BACnetDateTime;
	Log_DeviceObjectProperty	:BACnetDeviceObjectPropertyReference;
	Log_Interval					:WORD;
	COV_Resubscription_Interval:WORD;
	Client_COV_Increment		:BACnetClientCOV;
	Stop_When_Full				:BOOL;
	Buffer_Size					:DWORD;
	Log_Buffer					:ARRAY [0..MAX_Log_Buffer] OF BACnetLogRecord;
	Record_Count				:DWORD;
	Total_Record_Count			:DWORD;
	Notification_Threshold		:DWORD;
	Records_Since_Notification	:DWORD;
	Last_Notify_Record			:DWORD;
	Event_State					:BACnetEventState;
	Notification_Class			:WORD;
	Event_Enable					:BACnetEventTransitionBits;
	Acked_Transitions			:BACnetEventTransitionBits;
	Notify_Type					:BACnetNotifyType;
	Event_Time_Stamps			:ARRAY [1..3] OF BACnetTimeStamp;
END_STRUCT
END_TYPE

(* Data type in Datatypes *)
TYPE BACnetAccumulatorRecord :
STRUCT
	timestamp 			:BACnetDateTime;
	presentValue 			:WORD;
	accumulatedValue 	:WORD;
	accumulatorStatus	:AccumulatorStatus;
END_STRUCT
END_TYPE

(* Data type in Enumerationen *)
TYPE BACnetAction :(
	direct		:=0,
	reverse	:=1);
END_TYPE

(* Data type in Datatypes *)
TYPE BACnetActionCommand :
STRUCT
	deviceIdentifier		:BACnetObjectIdentifier;
	objectIdentifier		:BACnetObjectIdentifier;
	propertyIdentifier		:BACnetPropertyIdentifier;
	propertyArrayIndex	:WORD;
	priority					:WORD;
	postDelay				:WORD;
	quitOnFailure			:BOOL;
	writeSuccessful		:BOOL;
END_STRUCT
END_TYPE

(* Data type in Datatypes *)
TYPE BACnetActionList :
STRUCT
	BACnetAction : BACnetActionCommand;
END_STRUCT
END_TYPE

(* Data type in Datatypes *)
TYPE BACnetAddress :
STRUCT
	network_number	:WORD;
	mac_address		:BYTE;
END_STRUCT
END_TYPE

(* Data type in Datatypes *)
TYPE BACnetAddressBinding :
STRUCT
	deviceObjectIdentifier		:BACnetObjectIdentifier;
	deviceAddress			:BACnetAddress;
END_STRUCT
END_TYPE

(* Data type in Datatypes/internal *)
TYPE BACnetAny :
STRUCT
	CHOICE	:WORD;
	SIZE		:BYTE;
	VALUE		:ARRAY [0..254] OF BYTE;
END_STRUCT
END_TYPE

(* Data type in Enumerationen *)
TYPE BACnetBinaryPV :(
	inactive	:=0,
	active		:=1);
END_TYPE

(* Data type in Datatypes *)
TYPE BACnetCalendarEntry :
STRUCT
	CHOICE	:BYTE;
	VALUE		:ARRAY [0..21] OF BYTE;
END_STRUCT
END_TYPE

(* Data type in Datatypes *)
TYPE BACnetClientCOV :
STRUCT
	CHOICE	:BYTE;
	VALUE		:REAL;
END_STRUCT
END_TYPE

(* Data type in Datatypes *)
TYPE BACnetCOVSubscription :
STRUCT
	Recipient						:BACnetRecipientProcess;
	MonitoredPropertyReference	:BACnetObjectPropertyReference;
	IssueConfirmedNotifications	:BOOL;
	TimeRemaining				:WORD;
	COVIncrement				:REAL;
END_STRUCT
END_TYPE

(* Data type in Datatypes *)
TYPE BACnetDailySchedule :
STRUCT
	count			:WORD;
	day_schedule	:BACnetTimeValue;
END_STRUCT
END_TYPE

(* Data type in Datatypes *)
TYPE BACnetDateRange :
STRUCT
	StartDate		:DATE;
	endDate		:DATE;
END_STRUCT
END_TYPE

(* Data type in Datatypes *)
TYPE BACnetDateTime :
STRUCT
	BACnetDate	:DATE;
	BACnetTime	:TOD;
END_STRUCT
END_TYPE

(* Data type in Datatypes *)
TYPE BACnetDaysOfWeek :
STRUCT
	monday		:BOOL;
	tuesday		:BOOL;
	wednesday	:BOOL;
	thursday		:BOOL;
	friday			:BOOL;
	saturday		:BOOL;
	sunday		:BOOL;
END_STRUCT
END_TYPE

(* Data type in Datatypes *)
TYPE BACnetDestination :
STRUCT
	validDays						:BACnetDaysOfWeek;
	fromTime						:TIME;
	toTime							:TIME;
	recipient						:BACnetRecipient;
	processIdentifier				:DWORD;
	issueConfirmedNotifications	:BOOL;
	transitions						:BACnetEventTransitionBits;
END_STRUCT
END_TYPE

(* Data type in Datatypes *)
TYPE BACnetDeviceObjectPropertyReference :
STRUCT
	objectIdentifier		:BACnetObjectIdentifier;
	propertyIdentifier		:BACnetPropertyIdentifier;
	propertyArrayIndex	:WORD;
	deviceIdentifier		:BACnetObjectIdentifier;
	devicePresent			:BOOL;
END_STRUCT
END_TYPE

(* Data type in Datatypes *)
TYPE BACnetDeviceObjectPropertyValue :
STRUCT
	deviceIdentifier	: BACnetObjectIdentifier;
	objectIdentifier	: BACnetObjectIdentifier;
	propertyIdentifier 	: BACnetPropertyIdentifier;
	arrayIndex 			:WORD;
END_STRUCT
END_TYPE

(* Data type in Datatypes *)
TYPE BACnetDeviceObjectReference :
STRUCT
	deviceIdentifier	:BACnetObjectIdentifier;
	objectIdentifier	:BACnetObjectIdentifier;
	devicePresent		:BOOL;
END_STRUCT
END_TYPE

(* Data type in Enumerationen *)
TYPE BACnetDeviceStatus :(
	operational				:=0,
	operational_read_only	:=1,
	download_required		:=2,
	download_in_progress	:=3,
	non_operational			:=4,
	backup_in_progress		:=5);
END_TYPE

(* Data type in Enumerationen *)
TYPE BACnetEngineeringUnits :(
	square_meters	:=	0	,
	square_feet		:=	1	,
	milliamperes		:=	2	,
	amperes			:=	3	,
	ohms				:=	4	,
	volts				:=	5	,
	kilovolts			:=	6	,
	megavolts			:=	7	,
	volt_amperes		:=	8	,
	kilovolt_amperes	:=	9	,
	megavolt_amperes			:=	10	,
	volt_amperes_reactive		:=	11	,
	kilovolt_amperes_reactive	:=	12	,
	megavolt_amperes_reactive	:=	13	,
	degrees_phase				:=	14	,
	power_factor					:=	15	,
	joules							:=	16	,
	kilojoules					:=	17	,
	watt_hours				:=	18	,
	kilowatt_hours			:=	19	,
	btus						:=	20	,
	therms						:=	21	,
	ton_hours					:=	22	,
	joules_per_kilogram_dry_air		:=	23	,
	btus_per_pound_dry_air			:=	24	,
	cycles_per_hour					:=	25	,
	cycles_per_minute				:=	26	,
	hertz								:=	27	,
	grams_of_water_per_kilogram_dry_air	:=	28	,
	percent_relative_humidity				:=	29	,
	millimeters								:=	30	,
	meters			:=	31	,
	inches			:=	32	,
	feet			:=	33	,
	watts_per_square_foot		:=	34	,
	watts_per_square_meter		:=	35	,
	lumens						:=	36	,
	luxes							:=	37	,
	foot_candles				:=	38	,
	kilograms					:=	39	,
	pounds_mass			:=	40	,
	tons						:=	41	,
	kilograms_per_second	:=	42	,
	kilograms_per_minute	:=	43	,
	kilograms_per_hour		:=	44	,
	pounds_mass_per_minute	:=	45	,
	pounds_mass_per_hour	:=	46	,
	watts			:=	47	,
	kilowatts		:=	48	,
	megawatts	:=	49	,
	btus_per_hour	:=	50	,
	horsepower		:=	51	,
	tons_refrigeration	:=	52	,
	pascals			:=	53	,
	kilopascals		:=	54	,
	bars				:=	55	,
	pounds_force_per_square_inch	:=	56	,
	centimeters_of_water		:=	57	,
	inches_of_water			:=	58	,
	millimeters_of_mercury	:=	59	,
	centimeters_of_mercury	:=	60	,
	inches_of_mercury		:=	61	,
	degrees_Celsius			:=	62	,
	degrees_Kelvin			:=	63	,
	degrees_Fahrenheit		:=	64	,
	degree_days_Celsius	:=	65	,
	degree_days_Fahrenheit	:=	66	,
	years		:=	67	,
	months	:=	68	,
	weeks		:=	69	,
	days		:=	70	,
	hours		:=	71	,
	minutes	:=	72	,
	seconds	:=	73	,
	meters_per_second	:=	74	,
	kilometers_per_hour	:=	75	,
	feet_per_second		:=	76	,
	feet_per_minute		:=	77	,
	miles_per_hour		:=	78	,
	cubic_feet				:=	79	,
	cubic_meters			:=	80	,
	imperial_gallons		:=	81	,
	liters					:=	82	,
	us_gallons			:=	83	,
	cubic_feet_per_minute		:=	84	,
	cubic_meters_per_second	:=	85	,
	imperial_gallons_per_minute	:=	86	,
	liters_per_second				:=	87	,
	liters_per_minute					:=	88	,
	us_gallons_per_minute			:=	89	,
	degrees_angular					:=	90	,
	degrees_Celsius_per_hour		:=	91	,
	degrees_Celsius_per_minute	:=	92	,
	degrees_Fahrenheit_per_hour	:=	93	,
	degrees_Fahrenheit_per_minute	:=	94	,
	no_units				:=	95	,
	parts_per_million		:=	96	,
	parts_per_billion		:=	97	,
	percent				:=	98	,
	percent_per_second	:=	99	,
	per_minute			:=	100	,
	per_second			:=	101	,
	psi_per_degree_Fahrenheit	:=	102	,
	radians					:=	103	,
	revolutions_per_minute	:=	104	,
	currency1					:=	105	,
	currency2					:=	106	,
	currency3					:=	107	,
	currency4					:=	108	,
	currency5					:=	109	,
	currency6					:=	110	,
	currency7					:=	111	,
	currency8					:=	112	,
	currency9					:=	113	,
	currency10				:=	114	,
	square_inches			:=	115	,
	square_centimeters		:=	116	,
	btus_per_pound			:=	117	,
	centimeters				:=	118	,
	pounds_mass_per_second	:=	119	,
	delta_degrees_Fahrenheit	:=	120	,
	delta_degrees_Kelvin		:=	121	,
	kilohms					:=	122	,
	megohms					:=	123	,
	millivolts					:=	124	,
	kilojoules_per_kilogram	:=	125	,
	megajoules				:=	126	,
	joules_per_degree_Kelvin				:=	127	,
	joules_per_kilogram_degree_Kelvin	:=	128	,
	kilohertz			:=	129	,
	megahertz			:=	130	,
	per_hour			:=	131	,
	milliwatts			:=	132	,
	hectopascals		:=	133	,
	millibars			:=	134	,
	cubic_meters_per_hour	:=	135	,
	liters_per_hour			:=	136	,
	kilowatt_hours_per_square_meter	:=	137	,
	kilowatt_hours_per_square_foot		:=	138	,
	megajoules_per_square_meter		:=	139	,
	megajoules_per_square_foot		:=	140	,
	watts_per_square_meter_degree_kelvin	:=	141	,
	cubic_feet_per_second			:=	142	,
	percent_obscuration_per_foot	:=	143	,
	percent_obscuration_per_meter	:=	144	,
	milliohms							:=	145	,
	megawatt_hours					:=	146	,
	kilo_btus							:=	147	,
	mega_btus						:=	148	,
	kilojoules_per_kilogram_dry_air	:=	149	,
	megajoules_per_kilogram_dry_air	:=	150	,
	kilojoules_per_degree_Kelvin	:=	151	,
	megajoules_per_degree_Kelvin	:=	152	,
	newton							:=	153	,
	grams_per_second				:=	154	,
	grams_per_minute				:=	155	,
	tons_per_hour					:=	156	,
	kilo_btus_per_hour				:=	157	,
	hundredths_seconds				:=	158	,
	milliseconds						:=	159	,
	newton_meters					:=	160	,
	millimeters_per_second			:=	161	,
	millimeters_per_minute			:=	162	,
	meters_per_minute				:=	163	,
	meters_per_hour					:=	164	,
	cubic_meters_per_minute		:=	165	,
	meters_per_second_per_second	:=	166	,
	amperes_per_meter				:=	167	,
	amperes_per_square_meter	:=	168	,
	ampere_square_meters			:=	169	,
	farads								:=	170	,
	henrys								:=	171	,
	ohm_meters						:=	172	,
	siemens							:=	173	,
	siemens_per_meter				:=	174	,
	teslas								:=	175	,
	volts_per_degree_Kelvin			:=	176	,
	volts_per_meter					:=	177	,
	webers							:=	178	,
	candelas							:=	179	,
	candelas_per_square_meter	:=	180	,
	degrees_Kelvin_per_hour		:=	181	,
	degrees_Kelvin_per_minute		:=	182	,
	joule_seconds					:=	183	,
	radians_per_second				:=	184	,
	square_meters_per_Newton		:=	185	,
	kilograms_per_cubic_meter		:=	186	,
	newton_seconds					:=	187	,
	newtons_per_meter				:=	188	,
	watts_per_meter_per_degree_Kelvin	:=	189);

END_TYPE

(* Data type in Datatypes *)
TYPE BACnetEventParameter :
STRUCT
	CHOICE	:BYTE;
	VALUE		:ARRAY [0..20] OF BYTE;
END_STRUCT
END_TYPE

(* Data type in Enumerationen *)
TYPE BACnetEventState :(
	normal,
	fault1,
	offnormal,
	high_limit,
	low_limit,
	life_safety_alarm);

END_TYPE

(* Data type in Datatypes *)
TYPE BACnetEventTransitionBits :
STRUCT
	to_offnormal	:BOOL;
	to_fault		:BOOL;
	to_normal		:BOOL;
END_STRUCT
END_TYPE

(* Data type in Enumerationen *)
TYPE BACnetEventType :(
	change_OF_bitstring:=0,
	change_of_state:=1,
	change_of_value:=2,
	command_failure:=3,
	floating_limit:=4,
	out_of_range:=5,

	change_OF_life_safety:=8,
	extended:=9	,
	buffer_ready:=10,
	unsigned_range:=11);

END_TYPE

(* Data type in Enumerationen *)
TYPE BACnetFileAccessMethod :(
	record_access	:=0,
	stream_access	:=1);
END_TYPE

(* Data type in Enumerationen *)
TYPE BACnetLifeSafetyMode :(
	off							:=0,
	on							:=1,
	test						:=2,
	manned						:=3,
	unmanned					:=4,
	armed						:=5,
	disarmed					:=6,
	prearmed					:=7,
	slow						:=8,
	fast						:=9,
	disconnected				:=10,
	enabled						:=11,
	disabled					:=12,
	automatic_release_disabled	:=13,
	default						:=14);
END_TYPE

(* Data type in Enumerationen *)
TYPE BACnetLifeSafetyOperation :(
	none				:=0,
	silence				:=1,
	silence_audible		:=2,
	silence_visual		:=3,
	reset				:=4,
	reset_alarm			:=5,
	reset_fault			:=6,
	unsilence			:=7,
	unsilence_audible	:=8,
	unsilence_visual	:=9);
END_TYPE

(* Data type in Enumerationen *)
TYPE BACnetLifeSafetyState :(
	quiet				:=0,
	pre_alarm			:=1,
	alarm_LiveState		:=2,
	fault_LiveState		:=3,
	fault_pre_alarm		:=4,
	fault_alarm			:=5,
	NOT_ready			:=6,
	active_LiveState	:=7,
	tamper				:=8,
	test_alarm			:=9,
	test_active			:=10,
	test_fault			:=11,
	test_fault_alarm	:=12,
	holdup				:=13,
	duress				:=14,
	tamper_alarm		:=15,
	abnormal_LiveState	:=16,
	emergency_power		:=17,
	delayed				:=18,
	blocked				:=19,
	local_alarm			:=20,
	general_alarm		:=21,
	supervisory			:=22,
	test_supervisory	:=23);
END_TYPE

(* Data type in Datatypes *)
TYPE BACnetLimitEnable :
STRUCT
	lowLimitEnable		:BOOL;
	highLimitEnable		:BOOL;
END_STRUCT
END_TYPE

(* Data type in Datatypes/internal *)
TYPE BACnetLogDatum :
STRUCT
	CHOICE	:BYTE;
	VALUE		:ARRAY[0..3] OF BYTE;
END_STRUCT
END_TYPE

(* Data type in Datatypes *)
TYPE BACnetLogRecord :
STRUCT
	timestamp		:BACnetDateTime;
	logDatum		:BACnetLogDatum;
	statusFlags	:BACnetStatusFlags;
END_STRUCT
END_TYPE

(* Data type in Datatypes *)
TYPE BACnetLogStatus :
STRUCT
	log_disabled:BOOL;
	buffer_purged:BOOL;
END_STRUCT
END_TYPE

(* Data type in Enumerationen *)
TYPE BACnetMaintenance :(
	none_Maintenance			:=0,
	periodic_test				:=1,
	need_service_operational	:=2,
	need_service_inoperative	:=3);
END_TYPE

(* Data type in Datatypes *)
TYPE BACnetNotificationParameters :
STRUCT
	CHOICE:BYTE;
	VALUE:ARRAY [0..20] OF BYTE;
END_STRUCT
END_TYPE

(* Data type in Enumerationen *)
TYPE BACnetNotifyType :(
	alarm,
	event,
	ack_notification);
END_TYPE

(* Data type in Datatypes *)
TYPE BACnetObjectIdentifier :
STRUCT
	BACnetObjectType	:BACnetObjectType;
	Instance				:DINT;
END_STRUCT
END_TYPE

(* Data type in Datatypes *)
TYPE BACnetObjectPropertyReference :
STRUCT
	objectIdentifier	:BACnetObjectIdentifier;
	propertyIdentifier	:BACnetPropertyIdentifier;
	propertyArrayIndex	:WORD;
END_STRUCT
END_TYPE

(* Data type in Datatypes *)
TYPE BACnetObjectPropertyValue :
STRUCT
	objectIdentifier		: BACnetObjectIdentifier;
	propertyIdentifier 		: BACnetPropertyIdentifier;
	propertyArrayIndex 	:WORD;
	value					:BACnetAny;
	priority				 	:WORD;
END_STRUCT
END_TYPE

(* Data type in Enumerationen *)
TYPE BACnetObjectType :(
	analog_input		:=0,
	analog_output		:=1,
	analog_value		:=2,
	binary_input		:=3,
	binary_output		:=4,
	binary_value		:=5,
	calendar			:=6,
	command			:=7,
	device				:=8,
	event_enrollment	:=9,
	file					:=10,
	group				:=11,
	loop				:=12,
	multi_state_input	:=13,
	multi_state_output:=14,
	notification_class	:=15,
	program_			:=16,
	schedule			:=17,
	averaging			:=18,
	multi_state_value	:=19,
	trend_log			:=20,
	life_safety_point	:=21,
	life_safety_zone	:=22,
	accumulator		:=23,
	pulse_converter	:=24);
END_TYPE

(* Data type in Datatypes *)
TYPE BACnetObjectTypesSupported :
STRUCT
	analog_input		:BOOL;
	analog_output		:BOOL;
	analog_value		:BOOL;
	binary_input		:BOOL;
	binary_output		:BOOL;
	binary_value		:BOOL;
	calendar			:BOOL;
	command				:BOOL;
	device				:BOOL;
	event_enrollment 	:BOOL;
	file				:BOOL;
	group				:BOOL;
	loop				:BOOL;
	multi_state_input	:BOOL;
	multi_state_output	:BOOL;
	notification_class	:BOOL;
	BACnetprogram	:BOOL;
	schedule			:BOOL;
	averaging			:BOOL;
	multi_state_value	:BOOL;
	trend_LOG			:BOOL;
	life_safety_point	:BOOL;
	life_safety_zone	:BOOL;
	accumulator			:BOOL;
	pulse_converter		:BOOL;
END_STRUCT
END_TYPE

(* Data type in Datatypes/internal *)
TYPE BACnetPeriod :
STRUCT
	CHOICE	:BYTE;
	VALUE		:ARRAY[0..7] OF BYTE;
END_STRUCT
END_TYPE

(* Data type in Enumerationen *)
TYPE BACnetPolarity :(
	normal_Polarity	:=0,
	reverse_Polarity	:=1);
END_TYPE

(* Data type in Datatypes *)
TYPE BACnetPrescale :
STRUCT
	multiplier		:WORD;
	moduloDivide	:WORD;
END_STRUCT
END_TYPE

(* Data type in Datatypes *)
TYPE BACnetPriorityArray :
STRUCT
	PriorityArray:ARRAY[1..16] OF BACnetPriorityValue;
END_STRUCT
END_TYPE

(* Data type in Datatypes *)
TYPE BACnetPriorityValue :
STRUCT
	CHOICE	:BYTE;
	VALUE		:DWORD;
END_STRUCT
END_TYPE

(* Data type in Enumerationen *)
TYPE BACnetProgramError :(
	normal_Error	:=0,
	load_failed		:=1,
	internal		:=2,
	program_Error	:=3,
	other			:=4);
END_TYPE

(* Data type in Enumerationen *)
TYPE BACnetProgramRequest :(
	ready		:=0,
	load		:=1,
	run			:=2,
	halt		:=3,
	restart		:=4,
	unload		:=5);
END_TYPE

(* Data type in Enumerationen *)
TYPE BACnetProgramState :(
	idle		:=0,
	loading		:=1,
	running		:=2,
	waiting		:=3,
	halted		:=4,
	unloading	:=5);
END_TYPE

(* Data type in Enumerationen *)
TYPE BACnetPropertyIdentifier :(
	acked_transitions						:=0,
	ack_required							:=1,
	action_									:=2,
	action_text								:=3,
	active_text								:=4,
	active_vt_sessions						:=5,
	alarm_value								:=6,
	alarm_values							:=7,
	all										:=8,
	all_writes_successful					:=9,
	apdu_segment_timeout					:=10,
	apdu_timeout							:=11,
	application_software_version			:=12,
	archive									:=13,
	bias									:=14,
	change_of_state_count					:=15,
	change_of_state_time					:=16,
	notification_class_Identifier			:=17,
	the_property_in_this_place_was_deleted	:=18,
	controlled_variable_reference			:=19,
	controlled_variable_units				:=20,
	controlled_variable_value				:=21,
	cov_increment							:=22,
	date_list								:=23,
	daylight_savings_status					:=24,
	deadband								:=25,
	derivative_constant						:=26,
	derivative_constant_units				:=27,
	description								:=28,
	description_of_halt						:=29,
	device_address_binding					:=30,
	device_type								:=31,
	effective_period						:=32,
	elapsed_active_time						:=33,
	error_limit								:=34,
	event_enable							:=35,
	event_state								:=36,
	event_type								:=37,
	exception_schedule						:=38,
	fault_values							:=39,
	feedback_value							:=40,
	file_access_method						:=41,
	file_size								:=42,
	file_type								:=43,
	firmware_revision						:=44,
	high_limit_identifier					:=45,
	inactive_text							:=46,
	in_process								:=47,
	instance_of								:=48,
	integral_constant						:=49,
	integral_constant_units					:=50,
	issue_confirmed_notifications			:=51,
	limit_enable							:=52,
	list_of_group_members					:=53,
	list_of_object_property_references		:=54,
	list_of_session_keys					:=55,
	local_date								:=56,
	local_time								:=57,
	location								:=58,
	low_limit_identifier					:=59,
	manipulated_variable_reference			:=60,
	maximum_output							:=61,
	max_apdu_length_accepted				:=62,
	max_info_frames							:=63,
	max_master								:=64,
	max_pres_value							:=65,
	minimum_off_time						:=66,
	minimum_on_time							:=67,
	minimum_output							:=68,
	min_pres_value							:=69,
	model_name								:=70,
	modification_date						:=71,
	notify_type								:=72,
	number_of_APDU_retries					:=73,
	number_of_states						:=74,
	objectidentifier						:=75,
	object_list								:=76,
	object_name								:=77,
	object_property_reference				:=78,
	objecttype								:=79,
	optional								:=80,
	out_of_service_identifier				:=81,
	output_units							:=82,
	event_parameters						:=83,
	see_event_parameters					:=83,
	polarity								:=84,
	presentvalue							:=85,
	priority								:=86,
	priority_array							:=87,
	priority_for_writing					:=88,
	process_identifier						:=89,
	program_change							:=90,
	program_location						:=91,
	program_state							:=92,
	proportional_constant					:=93,
	proportional_constant_units				:=94,
	protocol_conformance_class				:=95,
	protocol_object_types_supported			:=96,
	protocol_services_supported				:=97,
	protocol_version						:=98,
	read_only_								:=99,
	reason_for_halt							:=100,
	recipient								:=101,
	recipient_list							:=102,
	reliability								:=103,
	relinquish_default						:=104,
	required								:=105,
	resolution								:=106,
	segmentation_supported					:=107,
	setpoint								:=108,
	setpoint_reference						:=109,
	state_text								:=110,
	status_flags							:=111,
	system_status							:=112,
	time_delay								:=113,
	time_of_active_time_reset				:=114,
	time_of_state_count_reset				:=115,
	time_synchronization_recipients			:=116,
	units									:=117,
	update_interval							:=118,
	utc_offset								:=119,
	vendor_identifier						:=120,
	vendor_name								:=121,
	vt_classes_supported					:=122,
	weekly_schedule							:=123,
	attempted_samples						:=124,
	average_value							:=125,
	buffer_size								:=126,
	client_cov_increment					:=127,
	cov_resubscription_interval				:=128,
	current_notify_time						:=129,
	event_time_stamps						:=130,
	log_buffer								:=131,
	log_device_object_property				:=132,
	log_enable								:=133,
	log_interval							:=134,
	maximum_value							:=135,
	minimum_value							:=136,
	notification_threshold					:=137,
	previous_notify_time					:=138,
	protocol_revision						:=139,
	records_since_notification				:=140,
	record_count							:=141,
	start_time								:=142,
	stop_time								:=143,
	stop_when_full							:=144,
	total_record_count						:=145,
	valid_samples							:=146,
	window_interval							:=147,
	window_samples							:=148,
	maximum_value_timestamp					:=149,
	minimum_value_timestamp					:=150,
	variance_value							:=151,
	active_cov_subscriptions				:=152,
	backup_failure_timeout					:=153,
	configuration_files						:=154,
	database_revision						:=155,
	direct_reading							:=156,
	last_restore_time						:=157,
	maintenance_required					:=158,
	member_of								:=159,
	mode									:=160,
	operation_expected						:=161,
	setting									:=162,
	silenced								:=163,
	tracking_value							:=164,
	zone_members							:=165,
	life_safety_alarm_values				:=166,
	max_segments_accepted					:=167,
	profile_name							:=168,
	auto_slave_discovery					:=169,
	manual_slave_address_binding			:=170,
	slave_address_binding					:=171,
	slave_proxy_enable						:=172,
	last_notify_record						:=173,
	schedule_default						:=174,
	accepted_modes							:=175,
	adjust_value							:=176,
	count									:=177,
	count_before_change						:=178,
	count_change_time						:=179,
	cov_period								:=180,
	input_reference							:=181,
	limit_monitoring_interval				:=182,
	logging_object							:=183,
	logging_record							:=184,
	prescale								:=185,
	pulse_rate								:=186,
	scale									:=187,
	scale_factor							:=188,
	update_time								:=189,
	value_before_change						:=190,
	value_set								:=191,
	value_change_time						:=192);
END_TYPE

(* Data type in Datatypes *)
TYPE BACnetPropertyReference :
STRUCT
	propertyIdentifier		: BACnetPropertyIdentifier;
	propertyArrayIndex	:WORD;
END_STRUCT
END_TYPE

(* Data type in Datatypes *)
TYPE BACnetPropertyStates :
STRUCT
	CHOICE:BYTE;
	VALUE:DWORD;
END_STRUCT
END_TYPE

(* Data type in Datatypes *)
TYPE BACnetPropertyValue :
STRUCT
	PropertyIdentifier 		:BACnetPropertyIdentifier;
	propertyArrayIndex	:WORD;
	value					:BACnetAny;
	priority					:WORD;
END_STRUCT
END_TYPE

(* Data type in Datatypes *)
TYPE BACnetRecipient :
STRUCT
	CHOICE	:BYTE;
	VALUE		:ARRAY [0..11] OF BYTE;
END_STRUCT
END_TYPE

(* Data type in Datatypes *)
TYPE BACnetRecipientProcess :
STRUCT
	recipient			:BACnetObjectIdentifier;
	processIdentifier	:DWORD;
END_STRUCT
END_TYPE

(* Data type in Enumerationen *)
TYPE BACnetReliability :(
	no_fault_detected,
	no_sensor,
	over_range,
	under_range,
	open_loop,
	shorted_loop,
	no_output,
	unreliable_other,
	process_error,
	multi_state_fault,
	configuration_error);
END_TYPE

(* Data type in Datatypes *)
TYPE BACnetResultFlags :
STRUCT
	first_item:BOOL;
	last_item:BOOL;
	more_items:BOOL;
END_STRUCT
END_TYPE

(* Data type in Datatypes *)
TYPE BACnetScale :

STRUCT
	CHOICE	: BYTE;
	VALUE		: ARRAY [0..3] OF BYTE;
END_STRUCT
END_TYPE

(* Data type in Enumerationen *)
TYPE BACnetSegmentation :(
	segmented_both		:=0,
	segmented_transmit	:=1,
	segmented_receive	:=2,
	no_segmentation		:=3);
END_TYPE

(* Data type in Datatypes *)
TYPE BACnetServicesSupported :
STRUCT
	acknowledgeAlarm				:BOOL;
	confirmedCOVNotification		:BOOL;
	confirmedEventNotification		:BOOL;
	getAlarmSummary				:BOOL;
	getEnrollmentSummary			:BOOL;
	subscribeCOV					:BOOL;
	atomicReadFile					:BOOL;
	atomicWriteFile					:BOOL;
	addListElement					:BOOL;
	removeListElement				:BOOL;
	createObject						:BOOL;
	deleteObject						:BOOL;
	readProperty						:BOOL;
	readPropertyConditional			:BOOL;
	readPropertyMultiple				:BOOL;
	writeProperty 						:BOOL;
	writePropertyMultiple				:BOOL;
	deviceCommunicationControl	:BOOL;
	confirmedPrivateTransfer			:BOOL;
	confirmedTextMessage			:BOOL;
	reinitializeDevice					:BOOL;
	vtOpen								:BOOL;
	vtClose							:BOOL;
	vtData								:BOOL;
	authenticate						:BOOL;
	requestKey						:BOOL;
	i_Am								:BOOL;
	i_Have								:BOOL;
	unconfirmedCOVNotification		:BOOL;
	unconfirmedEventNotification	:BOOL;
	unconfirmedPrivateTransfer		:BOOL;
	unconfirmedTextMessage		:BOOL;
	timeSynchronization				:BOOL;
	who_Has							:BOOL;
	who_Is							:BOOL;
	readRange						:BOOL;
	utcTimeSynchronization			:BOOL;
	lifeSafetyOperation				:BOOL;
	subscribeCOVProperty			:BOOL;
	getEventInformation				:BOOL;
END_STRUCT
END_TYPE

(* Data type in Datatypes *)
TYPE BACnetSessionKey :
STRUCT
	sessionKey	:BYTE;
	peerAddress	:BACnetAddress;
END_STRUCT
END_TYPE

(* Data type in Datatypes *)
TYPE BACnetSetpointReference :
STRUCT
	present				:BOOL;
	setpointReference	:BACnetObjectPropertyReference;
END_STRUCT
END_TYPE

(* Data type in Enumerationen *)
TYPE BACnetSilencedState :(
	unsilenced			:=0,
	audible_silenced	:=1,
	visible_silenced	:=2,
	all_silenced		:=3);
END_TYPE

(* Data type in Datatypes *)
TYPE BACnetSpecialEvent :
STRUCT
	choiceTag			:BYTE;
	period				:BACnetPeriod;
	listOfTimeValues	:ARRAY [0..MAX_Exception_Schedule] OF BACnetTimeValue;
	eventPriority		:BYTE;
END_STRUCT
END_TYPE

(* Data type in Datatypes *)
TYPE BACnetStatusFlags :
STRUCT
	in_alarm					:BOOL;
	fault						:BOOL;
	overridden_StatusFlage	:BOOL;
	out_of_service			:BOOL;
END_STRUCT
END_TYPE

(* Data type in Datatypes *)
TYPE BACnetTimeStamp :
STRUCT
	CHOICE	:BYTE;
	VALUE		:ARRAY [0..7] OF BYTE;
END_STRUCT
END_TYPE

(* Data type in Datatypes *)
TYPE BACnetTimeValue :
STRUCT
	TIME_	:TIME;
	value	:BACnetAny;
END_STRUCT
END_TYPE

(* Data type in Enumerationen *)
TYPE BACnetVTClass :(
	default_terminal	:=0,
	ansi_x3_64		:=1,
	dec_vt52			:=2,
	dec_vt100			:=3,
	dec_vt220			:=4,
	hp_700_94		:=5,
	ibm_3130			:=6);
END_TYPE

(* Data type in Datatypes *)
TYPE BACnetVTSession :
STRUCT
	local_vtSessionID		:BYTE;
	remote_vtSessionID	:BYTE;
	remote_vtAddress	:BACnetAddress;
END_STRUCT
END_TYPE

(* Data type in Datatypes *)
TYPE BACnetWeekNDay :
STRUCT
	month			:BYTE;
	weekOfMonth	:BYTE;
	dayOfWeek	:BYTE;
END_STRUCT
END_TYPE

(* Data type in Logger *)
TYPE en_Logger_ErrLev :
(
	EL_Log			:=0,
	EL_Wrn			:=1,
	EL_Alarm		:=2,
	EL_AlarmStop	:=3
);
END_TYPE

(* Data type in Logger *)
TYPE en_Logger_Status :
(
	S_Logger_UNKNOWN := 0,
	S_Logger_IDLE,
	S_Logger_WAITCONN,
	S_Logger_WAITTX,
	S_Logger_WAITRESP,
	S_Logger_ERROR
);
END_TYPE

(* Data type *)
TYPE en_SYS_Objects :
(
	EO_SYS		:=0,  (* PLC *)
	EO_VPN		:=1,  (* VPN *)
	EO_DOOR		:=2,  (* Door & access control *)

	EO_CAL		:=10, (* Caldaia *)
	EO_CIR		:=11, (* Circolatore *)
	EO_CRON		:=12, (* Crono-termostato *)
	EO_VRD		:=13, (* Valvola miscelatore pannelli *)
	EO_CTL		:=14, (* Contalitri *)
	EO_CTB		:=15, (* Contabilizzatore *)
	EO_TPV		:=16, (* Temperature probes values *)
	EO_PPV		:=17, (* Pressure probes values *)
	EO_PBV		:=18, (* Over-Pressure Alarms *)
	EO_TBV		:=19, (* Over-Temperature Alarms *)
	EO_PMV		:=20, (* Under-Pressure Alarms *)
	EO_GRU		:=21, (* Gruppo termico *)
	EO_PDC		:=22, (* Pompa di calore *)
	EO_SOL		:=23, (* Pannello solare termico *)
	EO_ESOL		:=24, (* Pannello solare fotovoltaico *)
	EO_GAS		:=25, (* Contatore GAS *)
	EO_PORT		:=26, (* Misuratore di portata *)
	EO_FPV		:=27, (* Flow probes values *)
	EO_ANZ		:=28, (* Analizzatore di rete *)
	EO_SCA		:=29, (* Signal Control Alarms *)
	EO_LUX		:=30, (* Base Illumination point *)
	EO_LUXM		:=31, (* Metered Illumination point *)
	EO_PSG		:=32, (* Sensore di passaggio *)
	EO_HVAC		:=33, (* Heating, Ventilating and Air Conditioning *)
	EO_HYGRV	:=34, (* Relative Humidity sensors value *)
	EO_COOV		:=35, (* Carbon Dioxide CO2 sensors value *)
	EO_INV		:=36, (* Inverter *)
	EO_STR		:=37, (* Smart string box *)

	EO_CIRD		:=39, (* Double CIR *)
	EO_ACS		:=40, (* Hot domestic water *)
	EO_FRG		:=41, (* Frigo *)
	EO_THER		:=42, (* Thermostat *)
	EO_CIRM		:=43, (* Modbus CIR *)
	EO_CIRDM	:=44, (* Modbus double CIR *)

	EO_ZGW			:=200,  (* ZigBee - Gateway *)
	EO_ZRM			:=201,	(* ZigBee - Repeater *)
	EO_ZREL			:=202,	(* ZigBee - Actuator rele *)
	EO_ZTHL			:=203,	(* ZigBee - Temperature Sensor *)

	EO_ASGW			:=250,	(* ASi - Gateway *)
	EO_ASCBI		:=251,	(* ASi - Input Board, Ciabatta *)

	EO_LON			:=1000, (* Bus - LON *)
	EO_MODBUS		:=1001, (* Bus - MODBUS *)
	EO_MBUS			:=1002, (* Bus - M-BUS *)
	EO_MODBUS_TCP	:=1003, (* Bus - MODBUS TCP *)

	EO_GENERIC		:=9000, (* Generic dataset *)
	EO_EXPO			:=9001 (* EXPO dataset *)
);
END_TYPE

(* Data type *)
TYPE en_SYS_Status :
(
	S_UNKNOWN  := 0,
	S_STARTUP,
	S_INIT_RTC,
	S_INIT_VAR,
	S_AUTOTEST,
	S_RUNNING,
	S_SHUTDOWN,
	S_HALT
);
END_TYPE

(* Data type in Datatypes *)
TYPE ReadAccessResult :  								(*Dieser Datentyp muss noch definiert werden!!!!*)
STRUCT
	ObjectIdentifier	:BACnetObjectIdentifier;
	Present_Value	:REAL;
	Reliability			:BACnetReliability;
	Description		:STRING(48);
END_STRUCT
END_TYPE

(* Data type in Datatypes *)
TYPE ReadAccessSpecification :
STRUCT
	objectIdentifier			:BACnetObjectIdentifier;
	listOfPropertyReferences	:ARRAY [0..MAX_listOfPropertyReferences] OF BACnetPropertyReference;
END_STRUCT
END_TYPE

(* Data type in Logger *)
TYPE typ_Logger :
STRUCT
	Status		: en_Logger_Status;

	SendReq		: BOOL;
	SendIdx		: DWORD;
	SendData	: ARRAY [0..MAX_SEND_TCP_CLIENT] OF BYTE;
	SendLen		: DINT;

	TData		: ARRAY [0..MAX_SEND_TCP_CLIENT] OF BYTE;
	TLen		: DINT;

	LastIdxPos	: DWORD;

	(* Temporary variables used by objects *)
	s1			: STRING(256);
	i1			: WORD;

END_STRUCT
END_TYPE

(* Data type *)
TYPE typ_SYS :
STRUCT
	Status			: en_SYS_Status;
	Warning			: BOOL;
	Alarm			: BOOL;
	AlarmStop		: BOOL;

	Time_LogString	: STRING;
	Time_Year		: WORD;
	Time_Month		: BYTE;
	Time_Day		: BYTE;
	Time_Hour		: BYTE;
	Time_Minute		: BYTE;

	Time_CT_DT		: DT;
	Time_CT_Day		: WORD;
	Time_CT_Quarter	: BYTE;

	LastLogs_Idx	: BYTE;
	LastLogs_Dat	: ARRAY[0..5] OF STRING;
	LastLogs_Msg	: ARRAY[0..5] OF STRING;

END_STRUCT
END_TYPE

(* Data type in Datatypes *)
TYPE WriteAccessSpecification :
STRUCT
	objectIdentifier			:BACnetObjectIdentifier;
	listOfPropertyReferences	:BACnetPropertyValue; 	(*Hier muss noch die Größe der Liste definiert werden*)
END_STRUCT
END_TYPE

(* POU PLC_PRG, ST *)
PROGRAM PLC_PRG
VAR
	Timer1: TON; (* Fast controls tick *)
	Timer2: TON; (* Plant control tick *)
	Timer3: TON; (* Logger timer *)

	i	:	INT;

	HMI_AggiornaLog: BOOL;

	F: BOOL;


	EseguiLog: BYTE;
	Ton_pausaTrig: TON;
END_VAR

VAR_INPUT
	RichiestaLogDaRemoto: BOOL;
END_VAR
(******************************************************************************
 ****                           MAIN TASK CODE                             ****
 ******************************************************************************

	Network setup:
		IP  = 192.168.100.2 | MSK = 255.255.255.0
		GW	= 192.168.100.1 | DNS = 192.168.100.1
		SNTP = 193.204.114.232 (3600s) ==> 192.168.100.3

*)

(*==============================*)
(*===== Main status machine ====*)
(*==============================*)


Main_Stm();

(*==============================*)
(*== Running cycle operations ==*)
(*==============================*)
(*
IF SYS.Status>S_INIT_VAR THEN
	(* Execute cycle processes *)
(*	CAL01.Heartbeat( CLIM:=CAL01_Clima );*)
	(* Execute LON process *)
(*	Module_1_PRG(); *)


END_IF
*)
(*==============================*)
(*== System cycle operations ===*)
(*==============================*)
(* Execute TCP processes *)
Logger_Proc();
Remote_Proc();
(* Update user led *)
(*USRLED_Update(); *) (*++++++++++++++  moreno +++++++++++++++++*)
(* Execute Cron Editor commands *)
(*CronEd(); *)
 
END_PROGRAM
ACTION Main_Stm:
	Sys.Status:=S_RUNNING;


CASE Sys.Status OF

	S_STARTUP:
		Sys.Status:=S_INIT_RTC;

	S_INIT_RTC:
		(* Check RTC and update from network *)
		RTC_Update();
		(* Check time *)
		IF Sys.Time_Year>2000  THEN
			Sys.Status:=S_INIT_VAR;
		END_IF

	S_INIT_VAR:
		LogEv(EL_Wrn,EO_SYS,0,1,CONCAT('System_startup_v',WORD_TO_STRING(Plant_SW_VER)));
		Sys.Status:=S_RUNNING;

	S_RUNNING:
		Timer1(IN:=NOT Timer1.Q,PT:=T#50ms);
		IF Timer1.Q THEN
			(* Update meters *)

			(* Update system checks *)
			SYS_Proc();
		END_IF

		Timer2(IN:=NOT Timer2.Q,PT:=T#500ms);
		IF Timer2.Q THEN
			(* Read current date/time *)
			RTC_Update();


			(* Recupero informazioni dagli analizatori di rete  *)


			ANZ01(					(* Generale  QE1   Sottorete OP11  - BsB_MulCab4_Cab4QE1 *)
					Voltage_L1_N:= -9999,
					Voltage_L2_N:= -9999,
					Voltage_L3_N:= -9999,
					Voltage_L1_L2:= PLC_BAC.BsB_MulCab4_Cab4QE1_Vtm,
					Voltage_L2_L3:= PLC_BAC.BsB_MulCab4_Cab4QE1_Vtm,
					Voltage_L3_L1:= PLC_BAC.BsB_MulCab4_Cab4QE1_Vtm,
					Frequency:= -9999,
					Current_L1:= PLC_BAC.BsB_MulCab4_Cab4QE1_Itm,
					Current_L2:= PLC_BAC.BsB_MulCab4_Cab4QE1_Itm,
					Current_L3:= PLC_BAC.BsB_MulCab4_Cab4QE1_Itm,
					Current_L1_Max:= -9999,
					Current_L2_Max:=-9999 ,
					Current_L3_Max:= -9999,
					Power_factor_L1:= PLC_BAC.BsB_MulCab4_Cab4QE1_PF,
					Power_factor_L2:= PLC_BAC.BsB_MulCab4_Cab4QE1_PF,
					Power_factor_L3:= PLC_BAC.BsB_MulCab4_Cab4QE1_PF,
					ActivePower:=PLC_BAC.BsB_MulCab4_Cab4QE1_P *1000,
					ActivePower_Avg:= PLC_BAC.BsB_MulCab4_Cab4QE1_P*1000,
					ActivePower_Max:=-9999 ,
					ReactivePower:= -9999,
					ReactivePower_Max:= -9999,
					kWh_Active_energy:= -9999,
					kVArh_Reactive_energy:= -9999,
					Cosphi_L1:=-9999 ,
					Cosphi_L2:=-9999 ,
					Cosphi_L3:=-9999 ,
					AllarmeNodo:= FALSE , (*PLC_BAC.BsB_MulCab4_Cab4QE1_AllCom, *)
					 );


			ANZ02(					(* Generale  QE2 Continità - Sottorete OP11  - BsB_MulCab4_Cab4QE2C *)
					Voltage_L1_N:= -9999,
					Voltage_L2_N:= -9999,
					Voltage_L3_N:= -9999,
					Voltage_L1_L2:= PLC_BAC.BsB_MulCab4_Cab4QE2C_Vtm,
					Voltage_L2_L3:= PLC_BAC.BsB_MulCab4_Cab4QE2C_Vtm,
					Voltage_L3_L1:= PLC_BAC.BsB_MulCab4_Cab4QE2C_Vtm,
					Frequency:= -9999,
					Current_L1:= PLC_BAC.BsB_MulCab4_Cab4QE2C_Itm,
					Current_L2:= PLC_BAC.BsB_MulCab4_Cab4QE2C_Itm,
					Current_L3:= PLC_BAC.BsB_MulCab4_Cab4QE2C_Itm,
					Current_L1_Max:= -9999,
					Current_L2_Max:=-9999 ,
					Current_L3_Max:= -9999,
					Power_factor_L1:= PLC_BAC.BsB_MulCab4_Cab4QE2C_PF,
					Power_factor_L2:= PLC_BAC.BsB_MulCab4_Cab4QE2C_PF,
					Power_factor_L3:= PLC_BAC.BsB_MulCab4_Cab4QE2C_PF,
					ActivePower:=PLC_BAC.BsB_MulCab4_Cab4QE2C_P *1000,
					ActivePower_Avg:= PLC_BAC.BsB_MulCab4_Cab4QE2C_P*1000,
					ActivePower_Max:=-9999 ,
					ReactivePower:= -9999,
					ReactivePower_Max:= -9999,
					kWh_Active_energy:= -9999,
					kVArh_Reactive_energy:= -9999,
					Cosphi_L1:=-9999 ,
					Cosphi_L2:=-9999 ,
					Cosphi_L3:=-9999 ,
					AllarmeNodo:=  FALSE , (*PLC_BAC.BsB_MulCab4_Cab4QE2C_AllCom,*)
					 );


			ANZ03(					(* Generale  QE2  - Sottorete OP11  - BsB_MulCab4_Cab4QE2P *)
					Voltage_L1_N:= -9999,
					Voltage_L2_N:= -9999,
					Voltage_L3_N:= -9999,
					Voltage_L1_L2:= PLC_BAC.BsB_MulCab4_Cab4QE2P_Vtm,
					Voltage_L2_L3:= PLC_BAC.BsB_MulCab4_Cab4QE2P_Vtm,
					Voltage_L3_L1:= PLC_BAC.BsB_MulCab4_Cab4QE2P_Vtm,
					Frequency:= -9999,
					Current_L1:= PLC_BAC.BsB_MulCab4_Cab4QE2P_Itm,
					Current_L2:= PLC_BAC.BsB_MulCab4_Cab4QE2P_Itm,
					Current_L3:= PLC_BAC.BsB_MulCab4_Cab4QE2P_Itm,
					Current_L1_Max:= -9999,
					Current_L2_Max:=-9999 ,
					Current_L3_Max:= -9999,
					Power_factor_L1:= PLC_BAC.BsB_MulCab4_Cab4QE2P_PF,
					Power_factor_L2:= PLC_BAC.BsB_MulCab4_Cab4QE2P_PF,
					Power_factor_L3:= PLC_BAC.BsB_MulCab4_Cab4QE2P_PF,
					ActivePower:=PLC_BAC.BsB_MulCab4_Cab4QE2P_P*1000 ,
					ActivePower_Avg:=PLC_BAC.BsB_MulCab4_Cab4QE2P_P*1000 ,
					ActivePower_Max:=-9999 ,
					ReactivePower:= -9999,
					ReactivePower_Max:= -9999,
					kWh_Active_energy:= -9999,
					kVArh_Reactive_energy:= -9999,
					Cosphi_L1:=-9999 ,
					Cosphi_L2:=-9999 ,
					Cosphi_L3:=-9999 ,
					AllarmeNodo:=  FALSE , (*PLC_BAC.BsB_MulCab4_Cab4QE2P_AllCom,*)
					 );

			ANZ04(					(* Gruppo  Frigorifero CHW01  - Sottorete OP22  - Mult_MulC_QEGF01 *)
					Voltage_L1_N:= -9999,
					Voltage_L2_N:= -9999,
					Voltage_L3_N:= -9999,
					Voltage_L1_L2:= PLC_BAC.Mult_MulC_QEGF01_Vtm,
					Voltage_L2_L3:= PLC_BAC.Mult_MulC_QEGF01_Vtm,
					Voltage_L3_L1:= PLC_BAC.Mult_MulC_QEGF01_Vtm,
					Frequency:= -9999,
					Current_L1:= PLC_BAC.Mult_MulC_QEGF01_Itm,
					Current_L2:= PLC_BAC.Mult_MulC_QEGF01_Itm,
					Current_L3:= PLC_BAC.Mult_MulC_QEGF01_Itm,
					Current_L1_Max:= -9999,
					Current_L2_Max:=-9999 ,
					Current_L3_Max:= -9999,
					Power_factor_L1:= PLC_BAC.Mult_MulC_QEGF01_PF,
					Power_factor_L2:= PLC_BAC.Mult_MulC_QEGF01_PF,
					Power_factor_L3:= PLC_BAC.Mult_MulC_QEGF01_PF,
					ActivePower:=PLC_BAC.Mult_MulC_QEGF01_P*1000 ,
					ActivePower_Avg:= PLC_BAC.Mult_MulC_QEGF01_P*1000,
					ActivePower_Max:=-9999 ,
					ReactivePower:= -9999,
					ReactivePower_Max:= -9999,
					kWh_Active_energy:= -9999,
					kVArh_Reactive_energy:= -9999,
					Cosphi_L1:=-9999.,
					Cosphi_L2:=-9999 ,
					Cosphi_L3:=-9999 ,
					AllarmeNodo:=  FALSE , (*PLC_BAC.Mult_MulC_QEGF01_AllCom,*)
					 );

			ANZ05(					(* Gruppo  Frigorifero CHW02  - Sottorete OP22  - Mult_MulC_QGGF02 *)
					Voltage_L1_N:= -9999,
					Voltage_L2_N:= -9999,
					Voltage_L3_N:= -9999,
					Voltage_L1_L2:= PLC_BAC.Mult_MulC_QGGF02_Vtm,
					Voltage_L2_L3:= PLC_BAC.Mult_MulC_QGGF02_Vtm,
					Voltage_L3_L1:= PLC_BAC.Mult_MulC_QGGF02_Vtm,
					Frequency:=-9999,
					Current_L1:= PLC_BAC.Mult_MulC_QGGF02_Itm,
					Current_L2:= PLC_BAC.Mult_MulC_QGGF02_Itm,
					Current_L3:= PLC_BAC.Mult_MulC_QGGF02_Itm,
					Current_L1_Max:= -9999,
					Current_L2_Max:=-9999 ,
					Current_L3_Max:= -9999,
					Power_factor_L1:= PLC_BAC.Mult_MulC_QGGF02_PF,
					Power_factor_L2:= PLC_BAC.Mult_MulC_QGGF02_PF,
					Power_factor_L3:= PLC_BAC.Mult_MulC_QGGF02_PF,
					ActivePower:=PLC_BAC.Mult_MulC_QGGF02_P *1000,
					ActivePower_Avg:= PLC_BAC.Mult_MulC_QGGF02_P*1000,
					ActivePower_Max:=-9999 ,
					ReactivePower:= -9999,
					ReactivePower_Max:= -9999,
					kWh_Active_energy:= -9999,
					kVArh_Reactive_energy:= -9999,
					Cosphi_L1:=-9999 ,
					Cosphi_L2:=-9999 ,
					Cosphi_L3:=-9999 ,
					AllarmeNodo:=  FALSE , (*PLC_BAC.Mult_MulC_QGGF02_AllCom,*)
					 );

			ANZ06(					(* Generale da trafo TR1 - Sottorette OP22 - Mult_QGBT02 *)
					Voltage_L1_N:= -9999,
					Voltage_L2_N:= -9999,
					Voltage_L3_N:= -9999,
					Voltage_L1_L2:= PLC_BAC.Mult_QGBT02_Vtm,
					Voltage_L2_L3:= PLC_BAC.Mult_QGBT02_Vtm,
					Voltage_L3_L1:= PLC_BAC.Mult_QGBT02_Vtm,
					Frequency:= -9999,
					Current_L1:= PLC_BAC.Mult_QGBT02_Itm,
					Current_L2:= PLC_BAC.Mult_QGBT02_Itm,
					Current_L3:= PLC_BAC.Mult_QGBT02_Itm,
					Current_L1_Max:= -9999,
					Current_L2_Max:= -9999 ,
					Current_L3_Max:= -9999,
					Power_factor_L1:= PLC_BAC.Mult_QGBT02_PF,
					Power_factor_L2:= PLC_BAC.Mult_QGBT02_PF,
					Power_factor_L3:= PLC_BAC.Mult_QGBT02_PF,
					ActivePower:=PLC_BAC.Mult_QGBT02_P*1000 ,
					ActivePower_Avg:= PLC_BAC.Mult_QGBT02_P*1000,
					ActivePower_Max:= -9999 ,
					ReactivePower:= -9999,
					ReactivePower_Max:= -9999,
					kWh_Active_energy:= -9999,
					kVArh_Reactive_energy:= -9999,
					Cosphi_L1:= -9999 ,
					Cosphi_L2:= -9999 ,
					Cosphi_L3:= -9999 ,
					AllarmeNodo:=  FALSE , (*PLC_BAC.Mult_QGBT02_AllCom,*)
					 );

			ANZ07(					(* Alimentazine Piastra 1 da QGBT - Sottorette OP22 - Mult_QGBT03 *)
					Voltage_L1_N:= -9999,
					Voltage_L2_N:= -9999,
					Voltage_L3_N:= -9999,
					Voltage_L1_L2:= PLC_BAC.Mult_QGBT03_Vtm,
					Voltage_L2_L3:= PLC_BAC.Mult_QGBT03_Vtm,
					Voltage_L3_L1:= PLC_BAC.Mult_QGBT03_Vtm,
					Frequency:= -9999,
					Current_L1:= PLC_BAC.Mult_QGBT03_Itm,
					Current_L2:= PLC_BAC.Mult_QGBT03_Itm,
					Current_L3:= PLC_BAC.Mult_QGBT03_Itm,
					Current_L1_Max:= -9999,
					Current_L2_Max:= -9999 ,
					Current_L3_Max:= -9999,
					Power_factor_L1:= PLC_BAC.Mult_QGBT03_PF,
					Power_factor_L2:= PLC_BAC.Mult_QGBT03_PF,
					Power_factor_L3:= PLC_BAC.Mult_QGBT03_PF,
					ActivePower:=PLC_BAC.Mult_QGBT03_P*1000 ,
					ActivePower_Avg:= PLC_BAC.Mult_QGBT03_P*1000,
					ActivePower_Max:= -9999 ,
					ReactivePower:= -9999,
					ReactivePower_Max:= -9999,
					kWh_Active_energy:= -9999,
					kVArh_Reactive_energy:= -9999,
					Cosphi_L1:= -9999 ,
					Cosphi_L2:= -9999 ,
					Cosphi_L3:= -9999 ,
					AllarmeNodo:=  FALSE , (*PLC_BAC.Mult_QGBT03_AllCom,*)
					 );

			ANZ08(					(* Generale da trafo TR3 - Sottorette OP22 - Mult_QGBT04 *)
					Voltage_L1_N:= -9999,
					Voltage_L2_N:= -9999,
					Voltage_L3_N:= -9999,
					Voltage_L1_L2:= PLC_BAC.Mult_QGBT04_Vtm,
					Voltage_L2_L3:= PLC_BAC.Mult_QGBT04_Vtm,
					Voltage_L3_L1:= PLC_BAC.Mult_QGBT04_Vtm,
					Frequency:= -9999,
					Current_L1:= PLC_BAC.Mult_QGBT04_Itm,
					Current_L2:= PLC_BAC.Mult_QGBT04_Itm,
					Current_L3:= PLC_BAC.Mult_QGBT04_Itm,
					Current_L1_Max:= -9999,
					Current_L2_Max:= -9999 ,
					Current_L3_Max:= -9999,
					Power_factor_L1:=PLC_BAC.Mult_QGBT04_PF,
					Power_factor_L2:= PLC_BAC.Mult_QGBT04_PF,
					Power_factor_L3:= PLC_BAC.Mult_QGBT04_PF,
					ActivePower:=PLC_BAC.Mult_QGBT04_P *1000,
					ActivePower_Avg:= PLC_BAC.Mult_QGBT04_P*1000,
					ActivePower_Max:= -9999 ,
					ReactivePower:= -9999,
					ReactivePower_Max:= -9999,
					kWh_Active_energy:= -9999,
					kVArh_Reactive_energy:= -9999,
					Cosphi_L1:= -9999 ,
					Cosphi_L2:= -9999 ,
					Cosphi_L3:= -9999 ,
					AllarmeNodo:=  FALSE , (* PLC_BAC.Mult_QGBT04_AllCom, *)
					 );

			ANZ09(					(* Grupo frigo  - Sottorette OP22 - Mult_QGBT07 *)
					Voltage_L1_N:= -9999,
					Voltage_L2_N:= -9999,
					Voltage_L3_N:= -9999,
					Voltage_L1_L2:= PLC_BAC.Mult_QGBT07_Vtm,
					Voltage_L2_L3:= PLC_BAC.Mult_QGBT07_Vtm,
					Voltage_L3_L1:= PLC_BAC.Mult_QGBT07_Vtm,
					Frequency:= -9999,
					Current_L1:= PLC_BAC.Mult_QGBT07_Itm,
					Current_L2:= PLC_BAC.Mult_QGBT07_Itm,
					Current_L3:= PLC_BAC.Mult_QGBT07_Itm,
					Current_L1_Max:= -9999,
					Current_L2_Max:= -9999 ,
					Current_L3_Max:= -9999,
					Power_factor_L1:= PLC_BAC.Mult_QGBT07_PF,
					Power_factor_L2:= PLC_BAC.Mult_QGBT07_PF,
					Power_factor_L3:= PLC_BAC.Mult_QGBT07_PF,
					ActivePower:=PLC_BAC.Mult_QGBT07_P*1000 ,
					ActivePower_Avg:= PLC_BAC.Mult_QGBT07_P*1000 ,
					ActivePower_Max:= -9999 ,
					ReactivePower:= -9999,
					ReactivePower_Max:= -9999,
					kWh_Active_energy:= -9999,
					kVArh_Reactive_energy:= -9999,
					Cosphi_L1:= -9999 ,
					Cosphi_L2:= -9999 ,
					Cosphi_L3:= -9999 ,
					AllarmeNodo:=  FALSE , (*PLC_BAC.Mult_QGBT07_AllCom, *)
					 );

			ANZ10(					(* Riserva futuro frigorifero  - Sottorette OP22 - Mult_QGBT08 *)
					Voltage_L1_N:= -9999,
					Voltage_L2_N:= -9999,
					Voltage_L3_N:= -9999,
					Voltage_L1_L2:= PLC_BAC.Mult_QGBT08_Vtm,
					Voltage_L2_L3:= PLC_BAC.Mult_QGBT08_Vtm,
					Voltage_L3_L1:= PLC_BAC.Mult_QGBT08_Vtm,
					Frequency:= -9999,
					Current_L1:= PLC_BAC.Mult_QGBT08_Itm,
					Current_L2:= PLC_BAC.Mult_QGBT08_Itm,
					Current_L3:= PLC_BAC.Mult_QGBT08_Itm,
					Current_L1_Max:= -9999,
					Current_L2_Max:= -9999 ,
					Current_L3_Max:= -9999,
					Power_factor_L1:=PLC_BAC.Mult_QGBT08_PF,
					Power_factor_L2:= PLC_BAC.Mult_QGBT08_PF,
					Power_factor_L3:= PLC_BAC.Mult_QGBT08_PF,
					ActivePower:=PLC_BAC.Mult_QGBT08_P*1000 ,
					ActivePower_Avg:= PLC_BAC.Mult_QGBT08_P*1000,
					ActivePower_Max:= -9999 ,
					ReactivePower:= -9999,
					ReactivePower_Max:= -9999,
					kWh_Active_energy:= -9999,
					kVArh_Reactive_energy:= -9999,
					Cosphi_L1:= -9999 ,
					Cosphi_L2:= -9999 ,
					Cosphi_L3:= -9999 ,
					AllarmeNodo:=  FALSE , (*PLC_BAC.Mult_QGBT08_AllCom, *)
					 );

			ANZ11(					(* Riserva  - Sottorette OP22 - Mult_QGBT09 *)
					Voltage_L1_N:= -9999,
					Voltage_L2_N:= -9999,
					Voltage_L3_N:= -9999,
					Voltage_L1_L2:= PLC_BAC.Mult_QGBT09_Vtm,
					Voltage_L2_L3:= PLC_BAC.Mult_QGBT09_Vtm,
					Voltage_L3_L1:= PLC_BAC.Mult_QGBT09_Vtm,
					Frequency:= -9999,
					Current_L1:= PLC_BAC.Mult_QGBT09_Itm,
					Current_L2:= PLC_BAC.Mult_QGBT09_Itm,
					Current_L3:= PLC_BAC.Mult_QGBT09_Itm,
					Current_L1_Max:= -9999,
					Current_L2_Max:= -9999 ,
					Current_L3_Max:= -9999,
					Power_factor_L1:= PLC_BAC.Mult_QGBT09_PF,
					Power_factor_L2:= PLC_BAC.Mult_QGBT09_PF,
					Power_factor_L3:= PLC_BAC.Mult_QGBT09_PF,
					ActivePower:=PLC_BAC.Mult_QGBT09_P *1000,
					ActivePower_Avg:= PLC_BAC.Mult_QGBT09_P*1000,
					ActivePower_Max:= -9999 ,
					ReactivePower:= -9999,
					ReactivePower_Max:= -9999,
					kWh_Active_energy:= -9999,
					kVArh_Reactive_energy:= -9999,
					Cosphi_L1:= -9999,
					Cosphi_L2:= -9999 ,
					Cosphi_L3:= -9999 ,
					AllarmeNodo:=  FALSE , (*PLC_BAC.Mult_QGBT09_AllCom, *)
					 );

			ANZ12(					(* Riserva  - Sottorette OP22 - Mult_QGBT10 *)
					Voltage_L1_N:= -9999,
					Voltage_L2_N:= -9999,
					Voltage_L3_N:= -9999,
					Voltage_L1_L2:= PLC_BAC.Mult_QGBT10_Vtm,
					Voltage_L2_L3:= PLC_BAC.Mult_QGBT10_Vtm,
					Voltage_L3_L1:= PLC_BAC.Mult_QGBT10_Vtm,
					Frequency:= -9999,
					Current_L1:= PLC_BAC.Mult_QGBT10_Itm,
					Current_L2:= PLC_BAC.Mult_QGBT10_Itm,
					Current_L3:= PLC_BAC.Mult_QGBT10_Itm,
					Current_L1_Max:= -9999,
					Current_L2_Max:= -9999 ,
					Current_L3_Max:= -9999,
					Power_factor_L1:= PLC_BAC.Mult_QGBT10_PF,
					Power_factor_L2:= PLC_BAC.Mult_QGBT10_PF,
					Power_factor_L3:= PLC_BAC.Mult_QGBT10_PF,
					ActivePower:=PLC_BAC.Mult_QGBT10_P*1000 ,
					ActivePower_Avg:= PLC_BAC.Mult_QGBT10_P*1000,
					ActivePower_Max:= -9999 ,
					ReactivePower:= -9999,
					ReactivePower_Max:= -9999,
					kWh_Active_energy:= -9999,
					kVArh_Reactive_energy:= -9999,
					Cosphi_L1:= -9999 ,
					Cosphi_L2:= -9999 ,
					Cosphi_L3:= -9999 ,
					AllarmeNodo:=  FALSE , (*PLC_BAC.Mult_QGBT10_AllCom,*)
					 );

			ANZ13(					(* Impianto Water Mist  - Sottorette OP22 - Mult_QGBT11 *)
					Voltage_L1_N:= -9999,
					Voltage_L2_N:= -9999,
					Voltage_L3_N:= -9999,
					Voltage_L1_L2:= PLC_BAC.Mult_QGBT11_Vtm,
					Voltage_L2_L3:= PLC_BAC.Mult_QGBT11_Vtm,
					Voltage_L3_L1:= PLC_BAC.Mult_QGBT11_Vtm,
					Frequency:= -9999,
					Current_L1:= PLC_BAC.Mult_QGBT11_Itm,
					Current_L2:= PLC_BAC.Mult_QGBT11_Itm,
					Current_L3:= PLC_BAC.Mult_QGBT11_Itm,
					Current_L1_Max:= -9999,
					Current_L2_Max:= -9999 ,
					Current_L3_Max:= -9999,
					Power_factor_L1:=PLC_BAC.Mult_QGBT11_PF,
					Power_factor_L2:= PLC_BAC.Mult_QGBT11_PF,
					Power_factor_L3:= PLC_BAC.Mult_QGBT11_PF,
					ActivePower:=PLC_BAC.Mult_QGBT11_P*1000 ,
					ActivePower_Avg:= PLC_BAC.Mult_QGBT11_P*1000,
					ActivePower_Max:= -9999 ,
					ReactivePower:= -9999,
					ReactivePower_Max:= -9999,
					kWh_Active_energy:= -9999,
					kVArh_Reactive_energy:= -9999,
					Cosphi_L1:= -9999 ,
					Cosphi_L2:= -9999 ,
					Cosphi_L3:= -9999 ,
					AllarmeNodo:=  FALSE , (*PLC_BAC.Mult_QGBT11_AllCom,*)
					 );

			ANZ14(					(* QP3 Piano terzo D  - Sottorette OP22 - Mult_QGBT12 *)
					Voltage_L1_N:= -9999,
					Voltage_L2_N:= -9999,
					Voltage_L3_N:= -9999,
					Voltage_L1_L2:= PLC_BAC.Mult_QGBT12_Vtm,
					Voltage_L2_L3:= PLC_BAC.Mult_QGBT12_Vtm,
					Voltage_L3_L1:= PLC_BAC.Mult_QGBT12_Vtm,
					Frequency:= -9999,
					Current_L1:= PLC_BAC.Mult_QGBT12_Itm,
					Current_L2:= PLC_BAC.Mult_QGBT12_Itm,
					Current_L3:= PLC_BAC.Mult_QGBT12_Itm,
					Current_L1_Max:= -9999,
					Current_L2_Max:= -9999 ,
					Current_L3_Max:= -9999,
					Power_factor_L1:= PLC_BAC.Mult_QGBT12_PF,
					Power_factor_L2:= PLC_BAC.Mult_QGBT12_PF,
					Power_factor_L3:= PLC_BAC.Mult_QGBT12_PF,
					ActivePower:=PLC_BAC.Mult_QGBT12_P*1000 ,
					ActivePower_Avg:= PLC_BAC.Mult_QGBT12_P*1000,
					ActivePower_Max:= -9999 ,
					ReactivePower:= -9999,
					ReactivePower_Max:= -9999,
					kWh_Active_energy:= -9999,
					kVArh_Reactive_energy:= -9999,
					Cosphi_L1:= -9999 ,
					Cosphi_L2:= -9999 ,
					Cosphi_L3:= -9999 ,
					AllarmeNodo:=  FALSE , (*PLC_BAC.Mult_QGBT12_AllCom,*)
					 );

			ANZ15(					(* QP2 Piano secondo  D  - Sottorette OP22 - Mult_QGBT13 *)
					Voltage_L1_N:= -9999,
					Voltage_L2_N:= -9999,
					Voltage_L3_N:= -9999,
					Voltage_L1_L2:= PLC_BAC.Mult_QGBT13_Vtm,
					Voltage_L2_L3:= PLC_BAC.Mult_QGBT13_Vtm,
					Voltage_L3_L1:= PLC_BAC.Mult_QGBT13_Vtm,
					Frequency:= -9999,
					Current_L1:= PLC_BAC.Mult_QGBT13_Itm,
					Current_L2:= PLC_BAC.Mult_QGBT13_Itm,
					Current_L3:= PLC_BAC.Mult_QGBT13_Itm,
					Current_L1_Max:= -9999,
					Current_L2_Max:= -9999 ,
					Current_L3_Max:= -9999,
					Power_factor_L1:= PLC_BAC.Mult_QGBT13_PF,
					Power_factor_L2:=PLC_BAC.Mult_QGBT13_PF,
					Power_factor_L3:=PLC_BAC.Mult_QGBT13_PF,
					ActivePower:=PLC_BAC.Mult_QGBT13_P *1000,
					ActivePower_Avg:= PLC_BAC.Mult_QGBT13_P*1000,
					ActivePower_Max:= -9999 ,
					ReactivePower:= -9999,
					ReactivePower_Max:= -9999,
					kWh_Active_energy:= -9999,
					kVArh_Reactive_energy:= -9999,
					Cosphi_L1:= -9999 ,
					Cosphi_L2:= -9999 ,
					Cosphi_L3:= -9999 ,
					AllarmeNodo:=  FALSE , (*PLC_BAC.Mult_QGBT13_AllCom,*)
					 );

			ANZ16(					(* QP1 Piano primo  D  - Sottorette OP22 - Mult_QGBT14 *)
					Voltage_L1_N:= -9999,
					Voltage_L2_N:= -9999,
					Voltage_L3_N:= -9999,
					Voltage_L1_L2:= PLC_BAC.Mult_QGBT14_Vtm,
					Voltage_L2_L3:= PLC_BAC.Mult_QGBT14_Vtm,
					Voltage_L3_L1:= PLC_BAC.Mult_QGBT14_Vtm,
					Frequency:= -9999,
					Current_L1:= PLC_BAC.Mult_QGBT14_Itm,
					Current_L2:= PLC_BAC.Mult_QGBT14_Itm,
					Current_L3:= PLC_BAC.Mult_QGBT14_Itm,
					Current_L1_Max:= -9999,
					Current_L2_Max:= -9999 ,
					Current_L3_Max:= -9999,
					Power_factor_L1:= PLC_BAC.Mult_QGBT14_PF,
					Power_factor_L2:=PLC_BAC.Mult_QGBT14_PF,
					Power_factor_L3:=PLC_BAC.Mult_QGBT14_PF,
					ActivePower:=PLC_BAC.Mult_QGBT14_P*1000 ,
					ActivePower_Avg:= PLC_BAC.Mult_QGBT14_P*1000,
					ActivePower_Max:= -9999 ,
					ReactivePower:= -9999,
					ReactivePower_Max:= -9999,
					kWh_Active_energy:= -9999,
					kVArh_Reactive_energy:= -9999,
					Cosphi_L1:= -9999 ,
					Cosphi_L2:= -9999 ,
					Cosphi_L3:= -9999 ,
					AllarmeNodo:=  FALSE , (*PLC_BAC.Mult_QGBT14_AllCom,*)
					 );

			ANZ17(					(* QPT Piano primo  D  - Sottorette OP22 - Mult_QGBT15 *)
					Voltage_L1_N:= -9999,
					Voltage_L2_N:= -9999,
					Voltage_L3_N:= -9999,
					Voltage_L1_L2:= PLC_BAC.Mult_QGBT15_Vtm,
					Voltage_L2_L3:= PLC_BAC.Mult_QGBT15_Vtm,
					Voltage_L3_L1:= PLC_BAC.Mult_QGBT15_Vtm,
					Frequency:= -9999,
					Current_L1:= PLC_BAC.Mult_QGBT15_Itm,
					Current_L2:= PLC_BAC.Mult_QGBT15_Itm,
					Current_L3:= PLC_BAC.Mult_QGBT15_Itm,
					Current_L1_Max:= -9999,
					Current_L2_Max:= -9999 ,
					Current_L3_Max:= -9999,
					Power_factor_L1:= PLC_BAC.Mult_QGBT15_PF,
					Power_factor_L2:=PLC_BAC.Mult_QGBT15_PF,
					Power_factor_L3:=PLC_BAC.Mult_QGBT15_PF,
					ActivePower:=PLC_BAC.Mult_QGBT15_P *1000,
					ActivePower_Avg:= PLC_BAC.Mult_QGBT15_P*1000,
					ActivePower_Max:= -9999 ,
					ReactivePower:= -9999,
					ReactivePower_Max:= -9999,
					kWh_Active_energy:= -9999,
					kVArh_Reactive_energy:= -9999,
					Cosphi_L1:= -9999 ,
					Cosphi_L2:= -9999 ,
					Cosphi_L3:= -9999 ,
					AllarmeNodo:=  FALSE , (*PLC_BAC.Mult_QGBT15_AllCom,*)
					 );

			ANZ18(					(* QP1 Piano interrato  D  - Sottorette OP22 - Mult_QGBT16 *)
					Voltage_L1_N:= -9999,
					Voltage_L2_N:= -9999,
					Voltage_L3_N:= -9999,
					Voltage_L1_L2:= PLC_BAC.Mult_QGBT16_Vtm,
					Voltage_L2_L3:= PLC_BAC.Mult_QGBT16_Vtm,
					Voltage_L3_L1:= PLC_BAC.Mult_QGBT16_Vtm,
					Frequency:= -9999,
					Current_L1:= PLC_BAC.Mult_QGBT16_Itm,
					Current_L2:= PLC_BAC.Mult_QGBT16_Itm,
					Current_L3:= PLC_BAC.Mult_QGBT16_Itm,
					Current_L1_Max:= -9999,
					Current_L2_Max:= -9999 ,
					Current_L3_Max:= -9999,
					Power_factor_L1:= PLC_BAC.Mult_QGBT16_PF,
					Power_factor_L2:=PLC_BAC.Mult_QGBT16_PF,
					Power_factor_L3:=PLC_BAC.Mult_QGBT16_PF,
					ActivePower:=PLC_BAC.Mult_QGBT16_P *1000,
					ActivePower_Avg:= PLC_BAC.Mult_QGBT16_P*1000,
					ActivePower_Max:= -9999 ,
					ReactivePower:= -9999,
					ReactivePower_Max:= -9999,
					kWh_Active_energy:= -9999,
					kVArh_Reactive_energy:= -9999,
					Cosphi_L1:= -9999 ,
					Cosphi_L2:= -9999 ,
					Cosphi_L3:= -9999 ,
					AllarmeNodo:=  FALSE , (*PLC_BAC.Mult_QGBT16_AllCom,*)
					 );

			ANZ19(					(* Alimentazione cabina ricevimento L1  - Sottorette OP22 - Mult_QGBT17 *)
					Voltage_L1_N:= -9999,
					Voltage_L2_N:= -9999,
					Voltage_L3_N:= -9999,
					Voltage_L1_L2:= PLC_BAC.Mult_QGBT17_Vtm,
					Voltage_L2_L3:= PLC_BAC.Mult_QGBT17_Vtm,
					Voltage_L3_L1:= PLC_BAC.Mult_QGBT17_Vtm,
					Frequency:= -9999,
					Current_L1:= PLC_BAC.Mult_QGBT17_Itm,
					Current_L2:= PLC_BAC.Mult_QGBT17_Itm,
					Current_L3:= PLC_BAC.Mult_QGBT17_Itm,
					Current_L1_Max:= -9999,
					Current_L2_Max:= -9999 ,
					Current_L3_Max:= -9999,
					Power_factor_L1:= PLC_BAC.Mult_QGBT17_PF,
					Power_factor_L2:=PLC_BAC.Mult_QGBT17_PF,
					Power_factor_L3:=PLC_BAC.Mult_QGBT17_PF,
					ActivePower:=PLC_BAC.Mult_QGBT17_P*1000 ,
					ActivePower_Avg:= PLC_BAC.Mult_QGBT17_P*1000,
					ActivePower_Max:= -9999 ,
					ReactivePower:= -9999,
					ReactivePower_Max:= -9999,
					kWh_Active_energy:= -9999,
					kVArh_Reactive_energy:= -9999,
					Cosphi_L1:= -9999 ,
					Cosphi_L2:= -9999 ,
					Cosphi_L3:= -9999 ,
					AllarmeNodo:=  FALSE , (*PLC_BAC.Mult_QGBT17_AllCom,*)
					 );

			ANZ20(					(* Alimentazione cabina ricevimento L12  - Sottorette OP22 - Mult_QGBT18 *)
					Voltage_L1_N:= -9999,
					Voltage_L2_N:= -9999,
					Voltage_L3_N:= -9999,
					Voltage_L1_L2:= PLC_BAC.Mult_QGBT18_Vtm,
					Voltage_L2_L3:= PLC_BAC.Mult_QGBT18_Vtm,
					Voltage_L3_L1:= PLC_BAC.Mult_QGBT18_Vtm,
					Frequency:= -9999,
					Current_L1:= PLC_BAC.Mult_QGBT18_Itm,
					Current_L2:= PLC_BAC.Mult_QGBT18_Itm,
					Current_L3:= PLC_BAC.Mult_QGBT18_Itm,
					Current_L1_Max:= -9999,
					Current_L2_Max:= -9999 ,
					Current_L3_Max:= -9999,
					Power_factor_L1:= PLC_BAC.Mult_QGBT18_PF,
					Power_factor_L2:=PLC_BAC.Mult_QGBT18_PF,
					Power_factor_L3:=PLC_BAC.Mult_QGBT18_PF,
					ActivePower:=PLC_BAC.Mult_QGBT18_P*1000 ,
					ActivePower_Avg:= PLC_BAC.Mult_QGBT18_P*1000,
					ActivePower_Max:= -9999 ,
					ReactivePower:= -9999,
					ReactivePower_Max:= -9999,
					kWh_Active_energy:= -9999,
					kVArh_Reactive_energy:= -9999,
					Cosphi_L1:= -9999 ,
					Cosphi_L2:= -9999 ,
					Cosphi_L3:= -9999 ,
					AllarmeNodo:=  FALSE , (*PLC_BAC.Mult_QGBT18_AllCom,*)
					 );

			ANZ21(					(* Sezione generale da UPS1  - Sottorette OP22 - Mult_QUPSO01 *)
					Voltage_L1_N:= -9999,
					Voltage_L2_N:= -9999,
					Voltage_L3_N:= -9999,
					Voltage_L1_L2:= PLC_BAC.Mult_QUPS01_Vtm,
					Voltage_L2_L3:= PLC_BAC.Mult_QUPS01_Vtm,
					Voltage_L3_L1:= PLC_BAC.Mult_QUPS01_Vtm,
					Frequency:= -9999,
					Current_L1:= PLC_BAC.Mult_QUPS01_Itm,
					Current_L2:= PLC_BAC.Mult_QUPS01_Itm,
					Current_L3:= PLC_BAC.Mult_QUPS01_Itm,
					Current_L1_Max:= -9999,
					Current_L2_Max:= -9999 ,
					Current_L3_Max:= -9999,
					Power_factor_L1:= PLC_BAC.Mult_QUPS01_PF,
					Power_factor_L2:=PLC_BAC.Mult_QUPS01_PF,
					Power_factor_L3:=PLC_BAC.Mult_QUPS01_PF,
					ActivePower:=PLC_BAC.Mult_QUPS01_P*1000 ,
					ActivePower_Avg:= PLC_BAC.Mult_QUPS01_P*1000,
					ActivePower_Max:= -9999 ,
					ReactivePower:= -9999,
					ReactivePower_Max:= -9999,
					kWh_Active_energy:= -9999,
					kVArh_Reactive_energy:= -9999,
					Cosphi_L1:= -9999 ,
					Cosphi_L2:= -9999 ,
					Cosphi_L3:= -9999 ,
					AllarmeNodo:=  FALSE , (*PLC_BAC.Mult_QUPS01_AllCom,*)
					 );

			ANZ22(					(* Sezionatore generale  - Sottorette OP22 - Mult_QUPSO02 *)
					Voltage_L1_N:= -9999,
					Voltage_L2_N:= -9999,
					Voltage_L3_N:= -9999,
					Voltage_L1_L2:= PLC_BAC.Mult_QUPS02_Vtm,
					Voltage_L2_L3:= PLC_BAC.Mult_QUPS02_Vtm,
					Voltage_L3_L1:= PLC_BAC.Mult_QUPS02_Vtm,
					Frequency:= -9999,
					Current_L1:= PLC_BAC.Mult_QUPS02_Itm,
					Current_L2:= PLC_BAC.Mult_QUPS02_Itm,
					Current_L3:= PLC_BAC.Mult_QUPS02_Itm,
					Current_L1_Max:= -9999,
					Current_L2_Max:= -9999 ,
					Current_L3_Max:= -9999,
					Power_factor_L1:= PLC_BAC.Mult_QUPS02_PF,
					Power_factor_L2:=PLC_BAC.Mult_QUPS02_PF,
					Power_factor_L3:=PLC_BAC.Mult_QUPS02_PF,
					ActivePower:=PLC_BAC.Mult_QUPS02_P*1000 ,
					ActivePower_Avg:= PLC_BAC.Mult_QUPS02_P*1000,
					ActivePower_Max:= -9999 ,
					ReactivePower:= -9999,
					ReactivePower_Max:= -9999,
					kWh_Active_energy:= -9999,
					kVArh_Reactive_energy:= -9999,
					Cosphi_L1:= -9999 ,
					Cosphi_L2:= -9999 ,
					Cosphi_L3:= -9999 ,
					AllarmeNodo:=  FALSE , (*PLC_BAC.Mult_QUPS02_AllCom,*)
					 );

			ANZ23(					(* Sezione generale da UPS2  - Sottorette OP22 - Mult_QUPSO03 *)
					Voltage_L1_N:= -9999,
					Voltage_L2_N:= -9999,
					Voltage_L3_N:= -9999,
					Voltage_L1_L2:= PLC_BAC.Mult_QUPS03_Vtm,
					Voltage_L2_L3:= PLC_BAC.Mult_QUPS03_Vtm,
					Voltage_L3_L1:= PLC_BAC.Mult_QUPS03_Vtm,
					Frequency:= -9999,
					Current_L1:= PLC_BAC.Mult_QUPS03_Itm,
					Current_L2:= PLC_BAC.Mult_QUPS03_Itm,
					Current_L3:= PLC_BAC.Mult_QUPS03_Itm,
					Current_L1_Max:= -9999,
					Current_L2_Max:= -9999 ,
					Current_L3_Max:= -9999,
					Power_factor_L1:= PLC_BAC.Mult_QUPS03_PF,
					Power_factor_L2:=PLC_BAC.Mult_QUPS03_PF,
					Power_factor_L3:=PLC_BAC.Mult_QUPS03_PF,
					ActivePower:=PLC_BAC.Mult_QUPS03_P*1000 ,
					ActivePower_Avg:= PLC_BAC.Mult_QUPS03_P*1000,
					ActivePower_Max:= -9999 ,
					ReactivePower:= -9999,
					ReactivePower_Max:= -9999,
					kWh_Active_energy:= -9999,
					kVArh_Reactive_energy:= -9999,
					Cosphi_L1:= -9999 ,
					Cosphi_L2:= -9999 ,
					Cosphi_L3:= -9999 ,
					AllarmeNodo:=  FALSE , (*PLC_BAC.Mult_QUPS03_AllCom,*)
					 );

			ANZ24(					(* QP3 sezione dialisi  - Sottorette OP22 - Mult_QUPSO04 *)
					Voltage_L1_N:= -9999,
					Voltage_L2_N:= -9999,
					Voltage_L3_N:= -9999,
					Voltage_L1_L2:= PLC_BAC.Mult_QUPS04_Vtm,
					Voltage_L2_L3:= PLC_BAC.Mult_QUPS04_Vtm,
					Voltage_L3_L1:= PLC_BAC.Mult_QUPS04_Vtm,
					Frequency:= -9999,
					Current_L1:= PLC_BAC.Mult_QUPS04_Itm,
					Current_L2:= PLC_BAC.Mult_QUPS04_Itm,
					Current_L3:= PLC_BAC.Mult_QUPS04_Itm,
					Current_L1_Max:= -9999,
					Current_L2_Max:= -9999 ,
					Current_L3_Max:= -9999,
					Power_factor_L1:= PLC_BAC.Mult_QUPS04_PF,
					Power_factor_L2:=PLC_BAC.Mult_QUPS04_PF,
					Power_factor_L3:=PLC_BAC.Mult_QUPS04_PF,
					ActivePower:=PLC_BAC.Mult_QUPS04_P*1000 ,
					ActivePower_Avg:= PLC_BAC.Mult_QUPS04_P*1000,
					ActivePower_Max:= -9999 ,
					ReactivePower:= -9999,
					ReactivePower_Max:= -9999,
					kWh_Active_energy:= -9999,
					kVArh_Reactive_energy:= -9999,
					Cosphi_L1:= -9999 ,
					Cosphi_L2:= -9999 ,
					Cosphi_L3:= -9999 ,
					AllarmeNodo:=  FALSE , (*PLC_BAC.Mult_QUPS04_AllCom,*)
					 );

			ANZ26(					(* Generale Villa Elios  - Sottorette OP23 - Mult1_QEPC *)
					Voltage_L1_N:= -9999,
					Voltage_L2_N:= -9999,
					Voltage_L3_N:= -9999,
					Voltage_L1_L2:= PLC_BAC.Mult1_QEPC_Vtm,
					Voltage_L2_L3:= PLC_BAC.Mult1_QEPC_Vtm,
					Voltage_L3_L1:= PLC_BAC.Mult1_QEPC_Vtm,
					Frequency:= -9999,
					Current_L1:= PLC_BAC.Mult1_QEPC_Itm,
					Current_L2:= PLC_BAC.Mult1_QEPC_Itm,
					Current_L3:= PLC_BAC.Mult1_QEPC_Itm,
					Current_L1_Max:= -9999,
					Current_L2_Max:= -9999 ,
					Current_L3_Max:= -9999,
					Power_factor_L1:= PLC_BAC.Mult1_QEPC_PF,
					Power_factor_L2:=PLC_BAC.Mult1_QEPC_PF,
					Power_factor_L3:=PLC_BAC.Mult1_QEPC_PF,
					ActivePower:=PLC_BAC.Mult1_QEPC_P*1000 ,
					ActivePower_Avg:= PLC_BAC.Mult1_QEPC_P*1000,
					ActivePower_Max:= -9999 ,
					ReactivePower:= -9999,
					ReactivePower_Max:= -9999,
					kWh_Active_energy:= -9999,
					kVArh_Reactive_energy:= -9999,
					Cosphi_L1:= -9999 ,
					Cosphi_L2:= -9999 ,
					Cosphi_L3:= -9999 ,
					AllarmeNodo:=  FALSE , (*PLC_BAC.Mult1_QEPC_AllCom, *)
					 );

			ANZ27(					(* Generale sez. preferenziale  - Sottorette OP23 - Mult1_QGBT05 *)
					Voltage_L1_N:= -9999,
					Voltage_L2_N:= -9999,
					Voltage_L3_N:= -9999,
					Voltage_L1_L2:= PLC_BAC.Mult1_QGBT05_Vtm,
					Voltage_L2_L3:= PLC_BAC.Mult1_QGBT05_Vtm,
					Voltage_L3_L1:= PLC_BAC.Mult1_QGBT05_Vtm,
					Frequency:= -9999,
					Current_L1:= PLC_BAC.Mult1_QGBT05_Itm,
					Current_L2:= PLC_BAC.Mult1_QGBT05_Itm,
					Current_L3:= PLC_BAC.Mult1_QGBT05_Itm,
					Current_L1_Max:= -9999,
					Current_L2_Max:= -9999 ,
					Current_L3_Max:= -9999,
					Power_factor_L1:= PLC_BAC.Mult1_QGBT05_PF,
					Power_factor_L2:=PLC_BAC.Mult1_QGBT05_PF,
					Power_factor_L3:=PLC_BAC.Mult1_QGBT05_PF,
					ActivePower:=PLC_BAC.Mult1_QGBT05_P*1000 ,
					ActivePower_Avg:= PLC_BAC.Mult1_QGBT05_P*1000,
					ActivePower_Max:= -9999 ,
					ReactivePower:= -9999,
					ReactivePower_Max:= -9999,
					kWh_Active_energy:= -9999,
					kVArh_Reactive_energy:= -9999,
					Cosphi_L1:= -9999 ,
					Cosphi_L2:= -9999 ,
					Cosphi_L3:= -9999 ,
					AllarmeNodo:=  FALSE , (*PLC_BAC.Mult1_QGBT05_AllCom,*)
					 );

			ANZ28(					(* generale G.E.  - Sottorette OP23 - Mult1_QGBT06 *)
					Voltage_L1_N:= -9999,
					Voltage_L2_N:= -9999,
					Voltage_L3_N:= -9999,
					Voltage_L1_L2:= PLC_BAC.Mult1_QGBT06_Vtm,
					Voltage_L2_L3:= PLC_BAC.Mult1_QGBT06_Vtm,
					Voltage_L3_L1:= PLC_BAC.Mult1_QGBT06_Vtm,
					Frequency:= -9999,
					Current_L1:= PLC_BAC.Mult1_QGBT06_Itm,
					Current_L2:= PLC_BAC.Mult1_QGBT06_Itm,
					Current_L3:= PLC_BAC.Mult1_QGBT06_Itm,
					Current_L1_Max:= -9999,
					Current_L2_Max:= -9999 ,
					Current_L3_Max:= -9999,
					Power_factor_L1:= PLC_BAC.Mult1_QGBT06_PF,
					Power_factor_L2:=PLC_BAC.Mult1_QGBT06_PF,
					Power_factor_L3:=PLC_BAC.Mult1_QGBT06_PF,
					ActivePower:=PLC_BAC.Mult1_QGBT06_P*1000 ,
					ActivePower_Avg:= PLC_BAC.Mult1_QGBT06_P*1000,
					ActivePower_Max:= -9999 ,
					ReactivePower:= -9999,
					ReactivePower_Max:= -9999,
					kWh_Active_energy:= -9999,
					kVArh_Reactive_energy:= -9999,
					Cosphi_L1:= -9999 ,
					Cosphi_L2:= -9999 ,
					Cosphi_L3:= -9999 ,
					AllarmeNodo:=  FALSE , (*PLC_BAC.Mult1_QGBT06_AllCom,*)
					 );

			ANZ29(					(* Gruppo frigo polivalente GP01  - Sottorette OP23 - Mult1_QGBT19 *)
					Voltage_L1_N:= -9999,
					Voltage_L2_N:= -9999,
					Voltage_L3_N:= -9999,
					Voltage_L1_L2:= PLC_BAC.Mult1_QGBT19_Vtm,
					Voltage_L2_L3:= PLC_BAC.Mult1_QGBT19_Vtm,
					Voltage_L3_L1:= PLC_BAC.Mult1_QGBT19_Vtm,
					Frequency:= -9999,
					Current_L1:= PLC_BAC.Mult1_QGBT19_Itm,
					Current_L2:= PLC_BAC.Mult1_QGBT19_Itm,
					Current_L3:= PLC_BAC.Mult1_QGBT19_Itm,
					Current_L1_Max:= -9999,
					Current_L2_Max:= -9999 ,
					Current_L3_Max:= -9999,
					Power_factor_L1:= PLC_BAC.Mult1_QGBT19_PF,
					Power_factor_L2:=PLC_BAC.Mult1_QGBT19_PF,
					Power_factor_L3:=PLC_BAC.Mult1_QGBT19_PF,
					ActivePower:=PLC_BAC.Mult1_QGBT19_P*1000 ,
					ActivePower_Avg:= PLC_BAC.Mult1_QGBT19_P*1000,
					ActivePower_Max:= -9999 ,
					ReactivePower:= -9999,
					ReactivePower_Max:= -9999,
					kWh_Active_energy:= -9999,
					kVArh_Reactive_energy:= -9999,
					Cosphi_L1:= -9999 ,
					Cosphi_L2:= -9999 ,
					Cosphi_L3:= -9999 ,
					AllarmeNodo:=  FALSE , (*PLC_BAC.Mult1_QGBT19_AllCom,*)
					 );

			ANZ30(					(* QP2 quadro piano 2  - Sottorette OP23 - Mult1_QGBT20 *)
					Voltage_L1_N:= -9999,
					Voltage_L2_N:= -9999,
					Voltage_L3_N:= -9999,
					Voltage_L1_L2:= PLC_BAC.Mult1_QGBT20_Vtm,
					Voltage_L2_L3:= PLC_BAC.Mult1_QGBT20_Vtm,
					Voltage_L3_L1:= PLC_BAC.Mult1_QGBT20_Vtm,
					Frequency:= -9999,
					Current_L1:= PLC_BAC.Mult1_QGBT20_Itm,
					Current_L2:= PLC_BAC.Mult1_QGBT20_Itm,
					Current_L3:= PLC_BAC.Mult1_QGBT20_Itm,
					Current_L1_Max:= -9999,
					Current_L2_Max:= -9999 ,
					Current_L3_Max:= -9999,
					Power_factor_L1:=PLC_BAC.Mult1_QGBT20_PF,
					Power_factor_L2:=PLC_BAC.Mult1_QGBT20_PF,
					Power_factor_L3:=PLC_BAC.Mult1_QGBT20_PF,
					ActivePower:=PLC_BAC.Mult1_QGBT20_P *1000,
					ActivePower_Avg:= PLC_BAC.Mult1_QGBT20_P*1000,
					ActivePower_Max:= -9999 ,
					ReactivePower:= -9999,
					ReactivePower_Max:= -9999,
					kWh_Active_energy:= -9999,
					kVArh_Reactive_energy:= -9999,
					Cosphi_L1:= -9999 ,
					Cosphi_L2:= -9999 ,
					Cosphi_L3:= -9999 ,
					AllarmeNodo:=  FALSE , (*PLC_BAC.Mult1_QGBT20_AllCom,*)
					 );

			ANZ31(					(* QP1 quadro piano 1  - Sottorette OP23 - Mult1_QGBT21 *)
					Voltage_L1_N:= -9999,
					Voltage_L2_N:= -9999,
					Voltage_L3_N:= -9999,
					Voltage_L1_L2:= PLC_BAC.Mult1_QGBT21_Vtm,
					Voltage_L2_L3:= PLC_BAC.Mult1_QGBT21_Vtm,
					Voltage_L3_L1:= PLC_BAC.Mult1_QGBT21_Vtm,
					Frequency:= -9999,
					Current_L1:= PLC_BAC.Mult1_QGBT21_Itm,
					Current_L2:= PLC_BAC.Mult1_QGBT21_Itm,
					Current_L3:= PLC_BAC.Mult1_QGBT21_Itm,
					Current_L1_Max:= -9999,
					Current_L2_Max:= -9999 ,
					Current_L3_Max:= -9999,
					Power_factor_L1:=PLC_BAC.Mult1_QGBT21_PF,
					Power_factor_L2:=PLC_BAC.Mult1_QGBT21_PF,
					Power_factor_L3:=PLC_BAC.Mult1_QGBT21_PF,
					ActivePower:=PLC_BAC.Mult1_QGBT21_P*1000 ,
					ActivePower_Avg:= PLC_BAC.Mult1_QGBT21_P*1000,
					ActivePower_Max:= -9999 ,
					ReactivePower:= -9999,
					ReactivePower_Max:= -9999,
					kWh_Active_energy:= -9999,
					kVArh_Reactive_energy:= -9999,
					Cosphi_L1:= -9999 ,
					Cosphi_L2:= -9999 ,
					Cosphi_L3:= -9999 ,
					AllarmeNodo:=  FALSE , (*PLC_BAC.Mult1_QGBT21_AllCom,*)
					 );

			ANZ32(					(* QPT quadro piano terra  - Sottorette OP23 - Mult1_QGBT22 *)
					Voltage_L1_N:= -9999,
					Voltage_L2_N:= -9999,
					Voltage_L3_N:= -9999,
					Voltage_L1_L2:= PLC_BAC.Mult1_QGBT22_Vtm,
					Voltage_L2_L3:= PLC_BAC.Mult1_QGBT22_Vtm,
					Voltage_L3_L1:= PLC_BAC.Mult1_QGBT22_Vtm,
					Frequency:= -9999,
					Current_L1:= PLC_BAC.Mult1_QGBT22_Itm,
					Current_L2:= PLC_BAC.Mult1_QGBT22_Itm,
					Current_L3:= PLC_BAC.Mult1_QGBT22_Itm,
					Current_L1_Max:= -9999,
					Current_L2_Max:= -9999 ,
					Current_L3_Max:= -9999,
					Power_factor_L1:=PLC_BAC.Mult1_QGBT22_PF,
					Power_factor_L2:=PLC_BAC.Mult1_QGBT22_PF,
					Power_factor_L3:=PLC_BAC.Mult1_QGBT22_PF,
					ActivePower:=PLC_BAC.Mult1_QGBT22_P*1000 ,
					ActivePower_Avg:= PLC_BAC.Mult1_QGBT22_P*1000,
					ActivePower_Max:= -9999 ,
					ReactivePower:= -9999,
					ReactivePower_Max:= -9999,
					kWh_Active_energy:= -9999,
					kVArh_Reactive_energy:= -9999,
					Cosphi_L1:= -9999 ,
					Cosphi_L2:= -9999 ,
					Cosphi_L3:= -9999 ,
					AllarmeNodo:=  FALSE , (*PLC_BAC.Mult1_QGBT22_AllCom,*)
					 );

			ANZ33(					(* QP1 quadro piano interrato - Sottorette OP23 - Mult1_QGBT23 *)
					Voltage_L1_N:= -9999,
					Voltage_L2_N:= -9999,
					Voltage_L3_N:= -9999,
					Voltage_L1_L2:= PLC_BAC.Mult1_QGBT23_Vtm,
					Voltage_L2_L3:= PLC_BAC.Mult1_QGBT23_Vtm,
					Voltage_L3_L1:= PLC_BAC.Mult1_QGBT23_Vtm,
					Frequency:= -9999,
					Current_L1:= PLC_BAC.Mult1_QGBT23_Itm,
					Current_L2:= PLC_BAC.Mult1_QGBT23_Itm,
					Current_L3:= PLC_BAC.Mult1_QGBT23_Itm,
					Current_L1_Max:= -9999,
					Current_L2_Max:= -9999 ,
					Current_L3_Max:= -9999,
					Power_factor_L1:= PLC_BAC.Mult1_QGBT23_PF,
					Power_factor_L2:=PLC_BAC.Mult1_QGBT23_PF,
					Power_factor_L3:=PLC_BAC.Mult1_QGBT23_PF,
					ActivePower:=PLC_BAC.Mult1_QGBT23_P*1000 ,
					ActivePower_Avg:= PLC_BAC.Mult1_QGBT23_P*1000,
					ActivePower_Max:= -9999 ,
					ReactivePower:= -9999,
					ReactivePower_Max:= -9999,
					kWh_Active_energy:= -9999,
					kVArh_Reactive_energy:= -9999,
					Cosphi_L1:= -9999 ,
					Cosphi_L2:= -9999 ,
					Cosphi_L3:= -9999 ,
					AllarmeNodo:=  FALSE , (*PLC_BAC.Mult1_QGBT23_AllCom,*)
					 );

			ANZ34(					(* QP3 quadro piano terzo - Sottorette OP23 - Mult1_QGBT24 *)
					Voltage_L1_N:= -9999,
					Voltage_L2_N:= -9999,
					Voltage_L3_N:= -9999,
					Voltage_L1_L2:= PLC_BAC.Mult1_QGBT24_Vtm,
					Voltage_L2_L3:= PLC_BAC.Mult1_QGBT24_Vtm,
					Voltage_L3_L1:= PLC_BAC.Mult1_QGBT24_Vtm,
					Frequency:= -9999,
					Current_L1:= PLC_BAC.Mult1_QGBT24_Itm,
					Current_L2:= PLC_BAC.Mult1_QGBT24_Itm,
					Current_L3:= PLC_BAC.Mult1_QGBT24_Itm,
					Current_L1_Max:= -9999,
					Current_L2_Max:= -9999 ,
					Current_L3_Max:= -9999,
					Power_factor_L1:= PLC_BAC.Mult1_QGBT24_PF,
					Power_factor_L2:=PLC_BAC.Mult1_QGBT24_PF,
					Power_factor_L3:=PLC_BAC.Mult1_QGBT24_PF,
					ActivePower:=PLC_BAC.Mult1_QGBT24_P *1000,
					ActivePower_Avg:= PLC_BAC.Mult1_QGBT24_P*1000,
					ActivePower_Max:= -9999 ,
					ReactivePower:= -9999,
					ReactivePower_Max:= -9999,
					kWh_Active_energy:= -9999,
					kVArh_Reactive_energy:= -9999,
					Cosphi_L1:= -9999 ,
					Cosphi_L2:= -9999 ,
					Cosphi_L3:= -9999 ,
					AllarmeNodo:=  FALSE , (*PLC_BAC.Mult1_QGBT24_AllCom,*)
					 );

			ANZ35(					(* Quadro centrale UTA copertura - Sottorette OP23 - Mult1_QGBT25 *)
					Voltage_L1_N:= -9999,
					Voltage_L2_N:= -9999,
					Voltage_L3_N:= -9999,
					Voltage_L1_L2:= PLC_BAC.Mult1_QGBT25_Vtm,
					Voltage_L2_L3:= PLC_BAC.Mult1_QGBT25_Vtm,
					Voltage_L3_L1:= PLC_BAC.Mult1_QGBT25_Vtm,
					Frequency:= -9999,
					Current_L1:= PLC_BAC.Mult1_QGBT25_Itm,
					Current_L2:= PLC_BAC.Mult1_QGBT25_Itm,
					Current_L3:= PLC_BAC.Mult1_QGBT25_Itm,
					Current_L1_Max:= -9999,
					Current_L2_Max:= -9999 ,
					Current_L3_Max:= -9999,
					Power_factor_L1:= PLC_BAC.Mult1_QGBT25_PF,
					Power_factor_L2:=PLC_BAC.Mult1_QGBT25_PF,
					Power_factor_L3:=PLC_BAC.Mult1_QGBT25_PF,
					ActivePower:=PLC_BAC.Mult1_QGBT25_P *1000,
					ActivePower_Avg:= PLC_BAC.Mult1_QGBT25_P*1000,
					ActivePower_Max:= -9999 ,
					ReactivePower:= -9999,
					ReactivePower_Max:= -9999,
					kWh_Active_energy:= -9999,
					kVArh_Reactive_energy:= -9999,
					Cosphi_L1:= -9999 ,
					Cosphi_L2:= -9999 ,
					Cosphi_L3:= -9999 ,
					AllarmeNodo:=  FALSE , (* PLC_BAC.Mult1_QGBT25_AllCom, *)
					 );

